// TIA Portal project "Flaconneuse" (V16)

(* hardware
DEVICE "Station S71500/ET200MP_1"  S7-1500 station
   slot 0: "Châssis_0"  Rack  6ES7 590-1***0-0AA0
   slot 0: "PM 70W 120/230VAC"  PM 70W 120/230VAC  6EP1332-4BA00
   slot 1: "PLC_1"  CPU 1511-1 PN  6ES7 511-1AK02-0AB0  V2.8
      slot 3: "Ecran CPU_1"  6ES7591-1AA00-0AA0
      slot 32768: "Interface PROFINET_1"  X1
         slot 32769: "Port_1"  X1 P1
         slot 32770: "Port_2"  X1 P2
      slot 34817: "Virtual CP interface port_1"  Virtual CP interface port  Virtual CP interface port
   slot 2: "DI 32x24VDC BA_1"  DI 32x24VDC BA  6ES7 521-1BL10-0AA0  V1.0
   slot 3: "DQ 32x24VDC/0.5A BA_1"  DQ 32x24VDC/0.5A BA  6ES7 522-1BL10-0AA0  V1.0
   slot 4: "CM 1542-5_1"  CM 1542-5  6GK7 542-5DX00-0XE0  V1.0
*)

// ===== PLC "PLC_1"  CPU 1511-1 PN =====

VAR_GLOBAL   // PLC tag table "Table de variables standard"
   "Marche cycle" AT %I0.0 : Bool;
   "Arret cycle" AT %I0.1 : Bool;
   "Selecteur sur Auto" AT %I0.3 : Bool;
   "Selecteur sur Manu" AT %I0.4 : Bool;
   "BP Manu" AT %I0.5 : Bool;
   "BP Purge" AT %I0.6 : Bool;
   "S1 pa" AT %I1.0 : Bool;   // Flacon en entree
   "S2 t0" AT %I1.1 : Bool;   // Verin de transfert rentre
   "S3 t1" AT %I1.2 : Bool;   // Verin de transfert sorti
   "S4 e1" AT %I1.3 : Bool;   // Verin d entrainement sorti
   "S5 i1" AT %I1.4 : Bool;   // Verin d indexage sorti
   "S6 p1" AT %I1.5 : Bool;   // Pompe sorti
   "S7 p0" AT %I1.6 : Bool;   // Pompe rentree
   "S8 r0" AT %I1.7 : Bool;   // Verin de vissage en bas
   "S9 r1" AT %I2.0 : Bool;   // Verin de vissage en haut
   "S10 b" AT %I2.1 : Bool;   // Flacon maintenu
   "S11 bour" AT %I2.2 : Bool;   // Bourage en sortie
   "S12 pr" AT %I2.3 : Bool;   // Presence remplissage
   "Voyant defaut" AT %Q0.0 : Bool;
   "EV1 T-" AT %Q0.1 : Bool;   // Rentrer verin transfert
   "EV2 T+" AT %Q0.2 : Bool;   // Sortir verin transfert
   "EV3 E-" AT %Q0.3 : Bool;   // Rentrer verin entrainement
   "EV4 I-" AT %Q0.4 : Bool;   // Rentrer verin indexage
   "EV5 P+" AT %Q0.5 : Bool;   // Sortir pompe
   "EV6 P-" AT %Q0.6 : Bool;   // Rentrer pompe
   "EV7 A" AT %Q0.7 : Bool;   // Commande arrivee liquide
   "EV8 J" AT %Q1.0 : Bool;   // Commande sortie liquide
   "EV9 B+" AT %Q1.1 : Bool;   // Maintenir flacon
   "EV10 R+" AT %Q1.2 : Bool;   // Descendre vissage
   "KM1" AT %Q1.4 : Bool;   // Moteur tapis
   "KM2" AT %Q1.5 : Bool;   // Moteur visseuse
   "IndexPlateau" AT %MW200 : Int;   // Les trois premiers bits de ce mot servent à savoir si il y a (ou non) un flacon sous chacun des postes
   "FM_FinPlateau" AT %M100.0 : Bool;
   "CI" AT %M120.0 : Bool;   // Condition initiales ok
   "DefautActif" AT %MW300 : Word;
END_VAR

DATA_BLOCK "X30_TournerPlateau_DB"   // DB1
{ S7_Optimized_Access := 'TRUE' }
VERSION : 0.1
// stored: InstanceOfName X30_TournerPlateau
"X30_TournerPlateau"
BEGIN
END_DATA_BLOCK

DATA_BLOCK "Sorties_DB"   // DB2
{ S7_Optimized_Access := 'TRUE' }
VERSION : 0.1
// stored: InstanceOfName Sorties
"Sorties"
BEGIN
END_DATA_BLOCK

DATA_BLOCK "X100_Remplir_DB"   // DB3
{ S7_Optimized_Access := 'TRUE' }
VERSION : 0.1
// stored: InstanceOfName X100_Remplir
"X100_Remplir"
BEGIN
END_DATA_BLOCK

DATA_BLOCK "X130_Visser_DB"   // DB4
{ S7_Optimized_Access := 'TRUE' }
VERSION : 0.1
// stored: InstanceOfName X130_Visser
"X130_Visser"
BEGIN
END_DATA_BLOCK

DATA_BLOCK "X160_Evacuer_DB"   // DB5
{ S7_Optimized_Access := 'TRUE' }
VERSION : 0.1
// stored: InstanceOfName X160_Evacuer
"X160_Evacuer"
BEGIN
END_DATA_BLOCK

DATA_BLOCK "X10_Conduite_DB"   // DB6
{ S7_Optimized_Access := 'TRUE' }
VERSION : 0.1
// stored: InstanceOfName X10_Conduite
"X10_Conduite"
BEGIN
END_DATA_BLOCK

DATA_BLOCK "X500_ModesDeMarche_DB"   // DB7
{ S7_Optimized_Access := 'TRUE' }
VERSION : 0.1
// stored: InstanceOfName X500_ModesDeMarche
"X500_ModesDeMarche"
BEGIN
END_DATA_BLOCK

DATA_BLOCK "GestionIndexPlateau_DB"   // DB8
{ S7_Optimized_Access := 'TRUE' }
VERSION : 0.1
// stored: InstanceOfName GestionIndexPlateau
"GestionIndexPlateau"
BEGIN
END_DATA_BLOCK

DATA_BLOCK "CondInitiales_DB"   // DB9
{ S7_Optimized_Access := 'TRUE' }
VERSION : 0.1
// stored: InstanceOfName CondInitiales
"CondInitiales"
BEGIN
END_DATA_BLOCK

DATA_BLOCK "defauts_DB"   // DB12
{ S7_Optimized_Access := 'TRUE' }
VERSION : 0.1
// stored: InstanceOfName defauts
"defauts"
BEGIN
END_DATA_BLOCK

// folder: System blocks/Program resources

DATA_BLOCK "IEC_Timer_0_DB"   // DB10
{ S7_Optimized_Access := 'TRUE' }
AUTHOR : Simatic
FAMILY : IEC
NAME : IEC_TMR
VERSION : 1.0
// stored: InstanceOfName IEC_TIMER
"IEC_TIMER"
BEGIN
END_DATA_BLOCK

DATA_BLOCK "IEC_Timer_0_DB_1"   // DB11
{ S7_Optimized_Access := 'TRUE' }
AUTHOR : Simatic
FAMILY : IEC
NAME : IEC_TMR
VERSION : 1.0
// stored: InstanceOfName IEC_TIMER
"IEC_TIMER"
BEGIN
END_DATA_BLOCK

// folder: (top level)

FUNCTION_BLOCK "X30_TournerPlateau"   // FB1, GRAPH_PLUS
{ S7_Optimized_Access := 'TRUE' }
VERSION : 0.1
   VAR_INPUT
      OFF_SQ : Bool := false;   // Désactiver le graphe
      INIT_SQ : Bool := false;   // Mettre le graphe à l'état initial
      ACK_EF : Bool := false;   // Acquitter toutes les erreurs et perturbations
      S_PREV : Bool := false;   // Afficher l'étape précédente dans le paramètre S_NO
      S_NEXT : Bool := false;   // Afficher l'étape suivante dans le paramètre S_NO
      SW_AUTO : Bool := false;   // Mode automatique
      SW_TAP : Bool := false;   // Mode semi-automatique/Activation de l'étape suivante avec transition
      SW_TOP : Bool := false;   // Mode semi-automatique/Ignorer la transition
      SW_MAN : Bool := false;   // Mode manuel
      S_SEL : Int := 0;   // Sélectionner l'étape à afficher dans S_NO
      S_ON : Bool := false;   // Activer l'étape figurant dans le paramètre S_NO
      S_OFF : Bool := false;   // Désactiver l'étape figurant dans le paramètre S_NO
      T_PUSH : Bool := false;   // Validation de commutation pour transition en mode semi-automatique
   END_VAR
   VAR_OUTPUT
      S_NO : Int := 0;   // Numéro d'étape
      S_MORE : Bool := false;   // Il existe d'autres étapes qui peuvent être affichées dans S_NO.
      S_ACTIVE : Bool := false;   // L'étape affichée dans le paramètre S_NO est activée
      ERR_FLT : Bool := false;   // Erreur groupée Interlock or Supervision
      AUTO_ON : Bool := false;   // Mode automatique activé
      TAP_ON : Bool := false;   // Mode semi-automatique/Etape avec transition activé
      TOP_ON : Bool := false;   // Mode semi-automatique/Ignorer la transition activé
      MAN_ON : Bool := false;   // Mode manuel activé
   END_VAR
   VAR
      HMI_INFO : Array[0..8] of UInt;
      IF_PAR : G7_IfParPlus_V6;
      RT_DATA : G7_RTDataPlus_V6;   // Plage de données interne
      Trans1 : G7_TransitionPlus_V6;   // Structure de la transition
      Trans2 : G7_TransitionPlus_V6;   // Structure de la transition
      Trans3 : G7_TransitionPlus_V6;   // Structure de la transition
      Trans4 : G7_TransitionPlus_V6;   // Structure de la transition
      Trans5 : G7_TransitionPlus_V6;   // Structure de la transition
      Trans6 : G7_TransitionPlus_V6;   // Structure de la transition
      Trans7 : G7_TransitionPlus_V6;   // Structure de la transition
      Trans8 : G7_TransitionPlus_V6;   // Structure de la transition
      Step30 : G7_StepPlus_V6;   // Structure de l'étape
      Step32 : G7_StepPlus_V6;   // Structure de l'étape
      Step34 : G7_StepPlus_V6;   // Structure de l'étape
      Step36 : G7_StepPlus_V6;   // Structure de l'étape
      Step38 : G7_StepPlus_V6;   // Structure de l'étape
      Step40 : G7_StepPlus_V6;   // Structure de l'étape
      Step42 : G7_StepPlus_V6;   // Structure de l'étape
      Step44 : G7_StepPlus_V6;   // Structure de l'étape
      SINI : Array[0..1] of USInt;
      LSTT : Array[0..7] of USInt;
      ATAJ : Array[0..7] of USInt;
      ATAB : Array[0..7] of USInt;
      PSTT : Array[0..7] of USInt;
      NSTT : Array[0..7] of USInt;
      ASSJ : Array[0..7] of USInt;
      ASSB : Array[0..7] of USInt;
      PTTS : Array[0..7] of USInt;
      NTTS : Array[0..7] of USInt;
      SW_SQTS : Array[0..7] of USInt;
      SWITCH : Array[0..0] of USInt;
      TVX : Array[0..1] of USInt;
      TTX : Array[0..1] of USInt;
      TSX : Array[0..1] of USInt;
      S00X : Array[0..1] of USInt;
      SOFFX : Array[0..1] of USInt;
      SONX : Array[0..1] of USInt;
      SAX : Array[0..1] of USInt;
      SERRX : Array[0..8] of USInt;
      SMX : Array[0..8] of USInt;
      S0X : Array[0..8] of USInt;
      S1X : Array[0..8] of USInt;
      IL_ALARM_INST : Diag_Alarm;
      SUP_ALARM_INST : Diag_Alarm;
      STEP_TIME_ALARM_INST : Diag_Alarm;
      IEC_TIMER_INST : IEC_TIMER;
      TRANSACTION_FLAG : Bool := false;
   END_VAR
   // SINI[0] := 2;
   // LSTT[0] := 255;
   // LSTT[1] := 255;
   // LSTT[2] := 255;
   // LSTT[3] := 255;
   // LSTT[4] := 255;
   // LSTT[5] := 255;
   // LSTT[6] := 255;
   // ATAJ[1] := 1;
   // ATAJ[2] := 2;
   // ATAJ[3] := 3;
   // ATAJ[4] := 4;
   // ATAJ[5] := 5;
   // ATAJ[6] := 6;
   // ATAJ[7] := 7;
   // ATAB[1] := 1;
   // ATAB[2] := 2;
   // ATAB[3] := 3;
   // ATAB[4] := 4;
   // ATAB[5] := 5;
   // ATAB[6] := 6;
   // ATAB[7] := 7;
   // PSTT[1] := 1;
   // PSTT[2] := 2;
   // PSTT[3] := 3;
   // PSTT[4] := 4;
   // PSTT[5] := 5;
   // PSTT[6] := 6;
   // PSTT[7] := 7;
   // NSTT[0] := 1;
   // NSTT[1] := 2;
   // NSTT[2] := 3;
   // NSTT[3] := 4;
   // NSTT[4] := 5;
   // NSTT[5] := 6;
   // NSTT[6] := 7;
   // ASSJ[1] := 1;
   // ASSJ[2] := 2;
   // ASSJ[3] := 3;
   // ASSJ[4] := 4;
   // ASSJ[5] := 5;
   // ASSJ[6] := 6;
   // ASSJ[7] := 7;
   // ASSB[1] := 1;
   // ASSB[2] := 2;
   // ASSB[3] := 3;
   // ASSB[4] := 4;
   // ASSB[5] := 5;
   // ASSB[6] := 6;
   // ASSB[7] := 7;
   // PTTS[0] := 255;
   // PTTS[2] := 1;
   // PTTS[3] := 2;
   // PTTS[4] := 3;
   // PTTS[5] := 4;
   // PTTS[6] := 5;
   // PTTS[7] := 6;
   // NTTS[1] := 1;
   // NTTS[2] := 2;
   // NTTS[3] := 3;
   // NTTS[4] := 4;
   // NTTS[5] := 5;
   // NTTS[6] := 6;
   // NTTS[7] := 7;
   // TVX[0] := 16#1;
   // TTX[0] := 16#1;
   // TSX[0] := 16#1;
   // S00X[0] := 16#1;
   // SOFFX[0] := 16#1;
   // SONX[0] := 16#1;
   // SAX[0] := 16#1;
   // SERRX[0] := 16#1;
   // SMX[0] := 16#1;
   // S0X[0] := 16#1;
   // S1X[0] := 16#1;
BEGIN
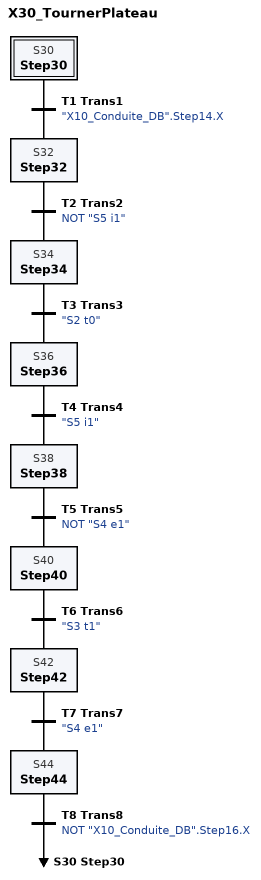
   // sequencer 1
   INITIAL_STEP Step30:   // S30, max time T#10S, warning time T#7S
   END_STEP
   TRANSITION Trans1 FROM Step30 TO Step32   // T1
      := "X10_Conduite_DB".Step14.X;
   END_TRANSITION
   STEP Step32:   // S32, max time T#10S, warning time T#7S
   END_STEP
   TRANSITION Trans2 FROM Step32 TO Step34   // T2: Vérin indexage rentré
      := NOT "S5 i1";
   END_TRANSITION
   STEP Step34:   // S34, max time T#10S, warning time T#7S
   END_STEP
   TRANSITION Trans3 FROM Step34 TO Step36   // T3: Vérin transfert rentré
      := "S2 t0";
   END_TRANSITION
   STEP Step36:   // S36, max time T#10S, warning time T#7S
   END_STEP
   TRANSITION Trans4 FROM Step36 TO Step38   // T4: vérin indexage sorti
      := "S5 i1";
   END_TRANSITION
   STEP Step38:   // S38, max time T#10S, warning time T#7S
   END_STEP
   TRANSITION Trans5 FROM Step38 TO Step40   // T5: Vérin entrainement rentré
      := NOT "S4 e1";
   END_TRANSITION
   STEP Step40:   // S40, max time T#10S, warning time T#7S
   END_STEP
   TRANSITION Trans6 FROM Step40 TO Step42   // T6: Vérin transfert sorti
      := "S3 t1";
   END_TRANSITION
   STEP Step42:   // S42, max time T#10S, warning time T#7S
   END_STEP
   TRANSITION Trans7 FROM Step42 TO Step44   // T7: Vérin entrainement sorti
      := "S4 e1";
   END_TRANSITION
   STEP Step44:   // S44, max time T#10S, warning time T#7S
   END_STEP
   TRANSITION Trans8 FROM Step44 TO Step30   // T8, jump
      := NOT "X10_Conduite_DB".Step16.X;
   END_TRANSITION
END_FUNCTION_BLOCK

FUNCTION_BLOCK "Sorties"   // FB2, LAD
{ S7_Optimized_Access := 'TRUE' }
VERSION : 0.1
BEGIN

REGION Network 1: Rentrer verin transfert
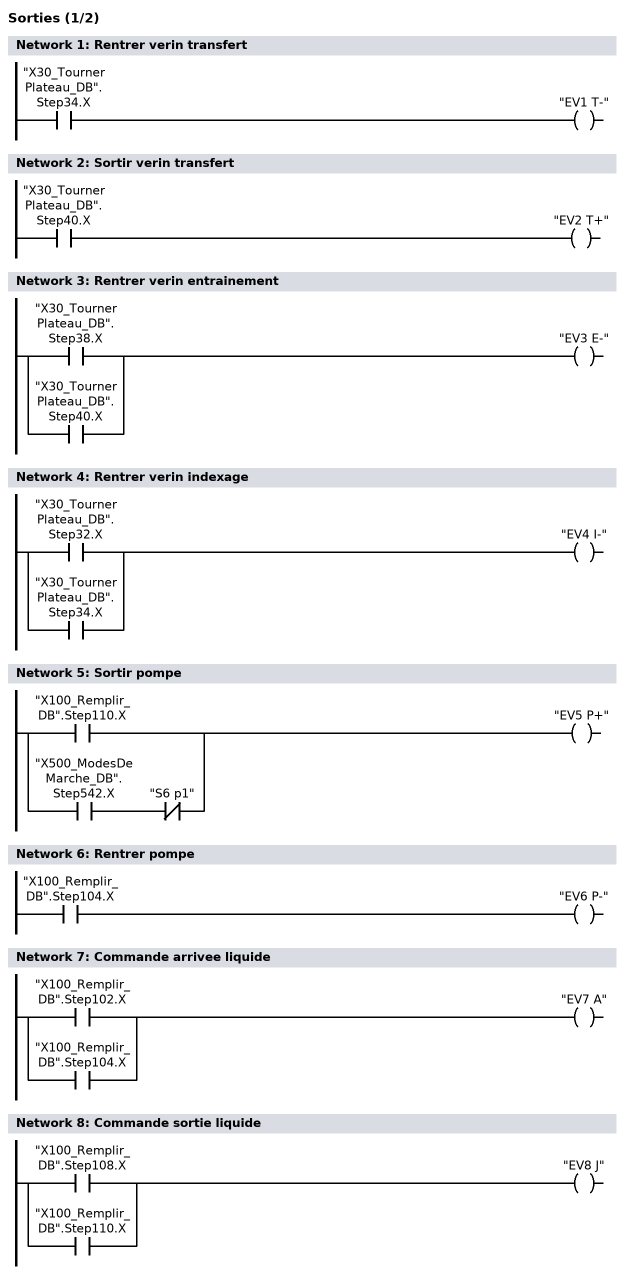
   RUNG wire#powerrail
      Contact( "X30_TournerPlateau_DB".Step34.X )
      Coil( "EV1 T-" )
   END_RUNG
   // the same network as SCL:
   "EV1 T-" := "X30_TournerPlateau_DB".Step34.X;
END_REGION

REGION Network 2: Sortir verin transfert
   RUNG wire#powerrail
      Contact( "X30_TournerPlateau_DB".Step40.X )
      Coil( "EV2 T+" )
   END_RUNG
   // the same network as SCL:
   "EV2 T+" := "X30_TournerPlateau_DB".Step40.X;
END_REGION

REGION Network 3: Rentrer verin entrainement
   RUNG wire#powerrail
      Contact( "X30_TournerPlateau_DB".Step38.X )
      wire#w1
      Coil( "EV3 E-" )
   END_RUNG
   RUNG wire#powerrail
      Contact( "X30_TournerPlateau_DB".Step40.X )
   END_RUNG wire#w1
   // the same network as SCL:
   "EV3 E-" := "X30_TournerPlateau_DB".Step38.X OR "X30_TournerPlateau_DB".Step40.X;
END_REGION

REGION Network 4: Rentrer verin indexage
   RUNG wire#powerrail
      Contact( "X30_TournerPlateau_DB".Step32.X )
      wire#w1
      Coil( "EV4 I-" )
   END_RUNG
   RUNG wire#powerrail
      Contact( "X30_TournerPlateau_DB".Step34.X )
   END_RUNG wire#w1
   // the same network as SCL:
   "EV4 I-" := "X30_TournerPlateau_DB".Step32.X OR "X30_TournerPlateau_DB".Step34.X;
END_REGION

REGION Network 5: Sortir pompe
   RUNG wire#powerrail
      Contact( "X100_Remplir_DB".Step110.X )
      wire#w1
      Coil( "EV5 P+" )
   END_RUNG
   RUNG wire#powerrail
      Contact( "X500_ModesDeMarche_DB".Step542.X )
      I_Contact( "S6 p1" )
   END_RUNG wire#w1
   // the same network as SCL:
   "EV5 P+" := "X100_Remplir_DB".Step110.X OR ("X500_ModesDeMarche_DB".Step542.X AND NOT "S6 p1");
END_REGION

REGION Network 6: Rentrer pompe
   RUNG wire#powerrail
      Contact( "X100_Remplir_DB".Step104.X )
      Coil( "EV6 P-" )
   END_RUNG
   // the same network as SCL:
   "EV6 P-" := "X100_Remplir_DB".Step104.X;
END_REGION

REGION Network 7: Commande arrivee liquide
   RUNG wire#powerrail
      Contact( "X100_Remplir_DB".Step102.X )
      wire#w1
      Coil( "EV7 A" )
   END_RUNG
   RUNG wire#powerrail
      Contact( "X100_Remplir_DB".Step104.X )
   END_RUNG wire#w1
   // the same network as SCL:
   "EV7 A" := "X100_Remplir_DB".Step102.X OR "X100_Remplir_DB".Step104.X;
END_REGION

REGION Network 8: Commande sortie liquide
   RUNG wire#powerrail
      Contact( "X100_Remplir_DB".Step108.X )
      wire#w1
      Coil( "EV8 J" )
   END_RUNG
   RUNG wire#powerrail
      Contact( "X100_Remplir_DB".Step110.X )
   END_RUNG wire#w1
   // the same network as SCL:
   "EV8 J" := "X100_Remplir_DB".Step108.X OR "X100_Remplir_DB".Step110.X;
END_REGION

REGION Network 9: Maintenir flacon
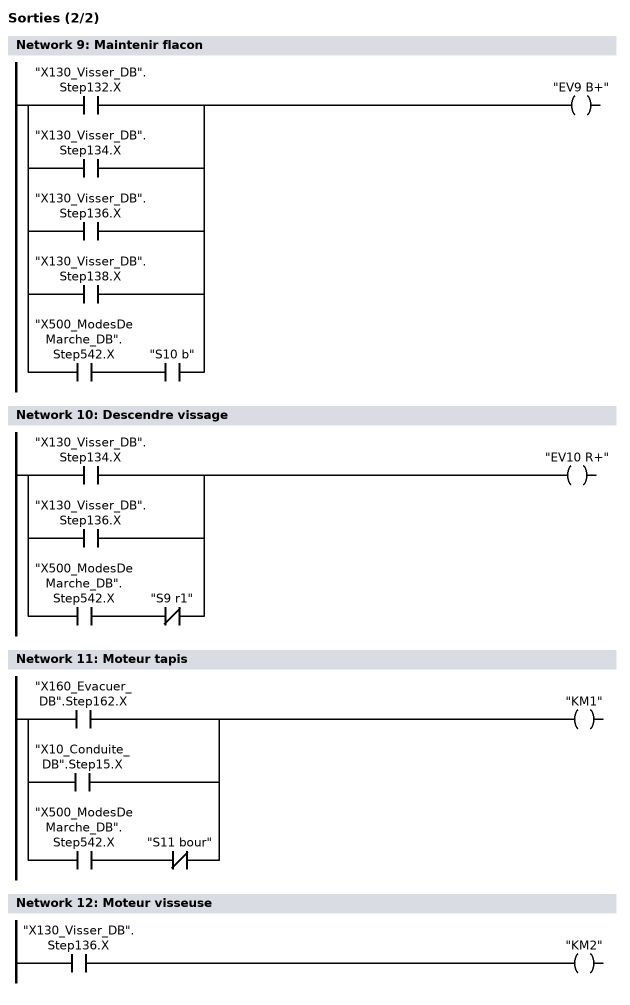
   RUNG wire#powerrail
      Contact( "X130_Visser_DB".Step132.X )
      wire#w1
      Coil( "EV9 B+" )
   END_RUNG
   RUNG wire#powerrail
      Contact( "X130_Visser_DB".Step134.X )
   END_RUNG wire#w1
   RUNG wire#powerrail
      Contact( "X130_Visser_DB".Step136.X )
   END_RUNG wire#w1
   RUNG wire#powerrail
      Contact( "X130_Visser_DB".Step138.X )
   END_RUNG wire#w1
   RUNG wire#powerrail
      Contact( "X500_ModesDeMarche_DB".Step542.X )
      Contact( "S10 b" )
   END_RUNG wire#w1
   // the same network as SCL:
   "EV9 B+" := "X130_Visser_DB".Step132.X OR "X130_Visser_DB".Step134.X OR "X130_Visser_DB".Step136.X OR "X130_Visser_DB".Step138.X OR ("X500_ModesDeMarche_DB".Step542.X AND "S10 b");
END_REGION

REGION Network 10: Descendre vissage
   RUNG wire#powerrail
      Contact( "X130_Visser_DB".Step134.X )
      wire#w1
      Coil( "EV10 R+" )
   END_RUNG
   RUNG wire#powerrail
      Contact( "X130_Visser_DB".Step136.X )
   END_RUNG wire#w1
   RUNG wire#powerrail
      Contact( "X500_ModesDeMarche_DB".Step542.X )
      I_Contact( "S9 r1" )
   END_RUNG wire#w1
   // the same network as SCL:
   "EV10 R+" := "X130_Visser_DB".Step134.X OR "X130_Visser_DB".Step136.X OR ("X500_ModesDeMarche_DB".Step542.X AND NOT "S9 r1");
END_REGION

REGION Network 11: Moteur tapis
   RUNG wire#powerrail
      Contact( "X160_Evacuer_DB".Step162.X )
      wire#w1
      Coil( "KM1" )
   END_RUNG
   RUNG wire#powerrail
      Contact( "X10_Conduite_DB".Step15.X )
   END_RUNG wire#w1
   RUNG wire#powerrail
      Contact( "X500_ModesDeMarche_DB".Step542.X )
      I_Contact( "S11 bour" )
   END_RUNG wire#w1
   // the same network as SCL:
   "KM1" := "X160_Evacuer_DB".Step162.X OR "X10_Conduite_DB".Step15.X OR ("X500_ModesDeMarche_DB".Step542.X AND NOT "S11 bour");
END_REGION

REGION Network 12: Moteur visseuse
   RUNG wire#powerrail
      Contact( "X130_Visser_DB".Step136.X )
      Coil( "KM2" )
   END_RUNG
   // the same network as SCL:
   "KM2" := "X130_Visser_DB".Step136.X;
END_REGION
END_FUNCTION_BLOCK

FUNCTION_BLOCK "X100_Remplir"   // FB3, GRAPH_PLUS
{ S7_Optimized_Access := 'TRUE' }
VERSION : 0.1
   VAR_INPUT
      OFF_SQ : Bool := false;   // Désactiver le graphe
      INIT_SQ : Bool := false;   // Mettre le graphe à l'état initial
      ACK_EF : Bool := false;   // Acquitter toutes les erreurs et perturbations
      S_PREV : Bool := false;   // Afficher l'étape précédente dans le paramètre S_NO
      S_NEXT : Bool := false;   // Afficher l'étape suivante dans le paramètre S_NO
      SW_AUTO : Bool := false;   // Mode automatique
      SW_TAP : Bool := false;   // Mode semi-automatique/Activation de l'étape suivante avec transition
      SW_TOP : Bool := false;   // Mode semi-automatique/Ignorer la transition
      SW_MAN : Bool := false;   // Mode manuel
      S_SEL : Int := 0;   // Sélectionner l'étape à afficher dans S_NO
      S_ON : Bool := false;   // Activer l'étape figurant dans le paramètre S_NO
      S_OFF : Bool := false;   // Désactiver l'étape figurant dans le paramètre S_NO
      T_PUSH : Bool := false;   // Validation de commutation pour transition en mode semi-automatique
   END_VAR
   VAR_OUTPUT
      S_NO : Int := 0;   // Numéro d'étape
      S_MORE : Bool := false;   // Il existe d'autres étapes qui peuvent être affichées dans S_NO.
      S_ACTIVE : Bool := false;   // L'étape affichée dans le paramètre S_NO est activée
      ERR_FLT : Bool := false;   // Erreur groupée Interlock or Supervision
      AUTO_ON : Bool := false;   // Mode automatique activé
      TAP_ON : Bool := false;   // Mode semi-automatique/Etape avec transition activé
      TOP_ON : Bool := false;   // Mode semi-automatique/Ignorer la transition activé
      MAN_ON : Bool := false;   // Mode manuel activé
   END_VAR
   VAR
      HMI_INFO : Array[0..8] of UInt;
      IF_PAR : G7_IfParPlus_V6;
      RT_DATA : G7_RTDataPlus_V6;   // Plage de données interne
      Trans2 : G7_TransitionPlus_V6;   // Structure de la transition
      Trans3 : G7_TransitionPlus_V6;   // Structure de la transition
      Trans4 : G7_TransitionPlus_V6;   // Structure de la transition
      Trans5 : G7_TransitionPlus_V6;   // Structure de la transition
      Trans6 : G7_TransitionPlus_V6;   // Structure de la transition
      Trans7 : G7_TransitionPlus_V6;   // Structure de la transition
      Trans8 : G7_TransitionPlus_V6;   // Structure de la transition
      Trans9 : G7_TransitionPlus_V6;   // Structure de la transition
      Step100 : G7_StepPlus_V6;   // Structure de l'étape
      Step102 : G7_StepPlus_V6;   // Structure de l'étape
      Step104 : G7_StepPlus_V6;   // Structure de l'étape
      Step106 : G7_StepPlus_V6;   // Structure de l'étape
      Step108 : G7_StepPlus_V6;   // Structure de l'étape
      Step110 : G7_StepPlus_V6;   // Structure de l'étape
      Step112 : G7_StepPlus_V6;   // Structure de l'étape
      SINI : Array[0..1] of USInt;
      LSTT : Array[0..7] of USInt;
      ATAJ : Array[0..7] of USInt;
      ATAB : Array[0..7] of USInt;
      PSTT : Array[0..7] of USInt;
      NSTT : Array[0..7] of USInt;
      ASSJ : Array[0..6] of USInt;
      ASSB : Array[0..6] of USInt;
      PTTS : Array[0..6] of USInt;
      NTTS : Array[0..6] of USInt;
      SW_SQTS : Array[0..6] of USInt;
      SWITCH : Array[0..1] of USInt;
      TVX : Array[0..3] of USInt;
      TTX : Array[0..3] of USInt;
      TSX : Array[0..1] of USInt;
      S00X : Array[0..1] of USInt;
      SOFFX : Array[0..1] of USInt;
      SONX : Array[0..1] of USInt;
      SAX : Array[0..1] of USInt;
      SERRX : Array[0..7] of USInt;
      SMX : Array[0..7] of USInt;
      S0X : Array[0..7] of USInt;
      S1X : Array[0..7] of USInt;
      IL_ALARM_INST : Diag_Alarm;
      SUP_ALARM_INST : Diag_Alarm;
      STEP_TIME_ALARM_INST : Diag_Alarm;
      IEC_TIMER_INST : IEC_TIMER;
      TRANSACTION_FLAG : Bool := false;
   END_VAR
   // SINI[0] := 2;
   // LSTT[0] := 255;
   // LSTT[1] := 255;
   // LSTT[2] := 255;
   // LSTT[3] := 255;
   // LSTT[4] := 255;
   // LSTT[6] := 255;
   // ATAJ[1] := 1;
   // ATAJ[2] := 2;
   // ATAJ[3] := 3;
   // ATAJ[4] := 6;
   // ATAJ[5] := 5;
   // ATAJ[6] := 4;
   // ATAB[1] := 1;
   // ATAB[2] := 2;
   // ATAB[3] := 3;
   // ATAB[4] := 4;
   // ATAB[5] := 5;
   // ATAB[6] := 7;
   // PSTT[1] := 2;
   // PSTT[2] := 3;
   // PSTT[3] := 4;
   // PSTT[4] := 5;
   // PSTT[5] := 6;
   // NSTT[7] := 1;
   // NSTT[0] := 2;
   // NSTT[1] := 3;
   // NSTT[2] := 4;
   // NSTT[3] := 5;
   // NSTT[4] := 6;
   // NSTT[6] := 6;
   // ASSJ[1] := 1;
   // ASSJ[2] := 2;
   // ASSJ[3] := 3;
   // ASSJ[4] := 4;
   // ASSJ[5] := 5;
   // ASSJ[6] := 6;
   // ASSB[1] := 1;
   // ASSB[2] := 2;
   // ASSB[3] := 3;
   // ASSB[4] := 4;
   // ASSB[5] := 5;
   // ASSB[6] := 6;
   // PTTS[0] := 255;
   // NTTS[0] := 7;
   // PTTS[3] := 1;
   // PTTS[4] := 2;
   // PTTS[5] := 3;
   // PTTS[6] := 4;
   // SW_SQTS[1] := 1;
   // NTTS[2] := 1;
   // NTTS[3] := 2;
   // NTTS[4] := 3;
   // NTTS[5] := 4;
   // NTTS[6] := 5;
   // TVX[0] := 16#1;
   // TTX[0] := 16#1;
   // TSX[0] := 16#1;
   // S00X[0] := 16#1;
   // SOFFX[0] := 16#1;
   // SONX[0] := 16#1;
   // SAX[0] := 16#1;
   // SERRX[0] := 16#1;
   // SMX[0] := 16#1;
   // S0X[0] := 16#1;
   // S1X[0] := 16#1;
   // LSTT[7] := 255;
   // ATAJ[7] := 7;
   // ATAB[7] := 6;
   // PSTT[0] := 1;
   // PTTS[1] := 7;
   // SW_SQTS[2] := 1;
   // SW_SQTS[3] := 1;
   // SW_SQTS[4] := 1;
   // SW_SQTS[5] := 1;
   // SW_SQTS[6] := 2;
BEGIN
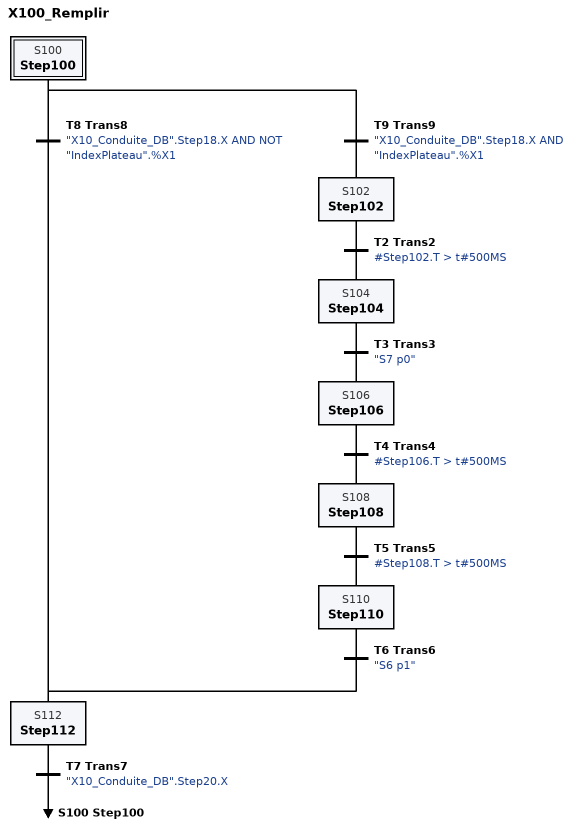
   // sequencer 1
   INITIAL_STEP Step100:   // S100, max time T#10S, warning time T#7S
   END_STEP
   TRANSITION Trans8 FROM Step100 TO Step112   // T8
      := "X10_Conduite_DB".Step18.X AND NOT "IndexPlateau".%X1;
   END_TRANSITION
   TRANSITION Trans9 FROM Step100 TO Step102   // T9
      := "X10_Conduite_DB".Step18.X AND "IndexPlateau".%X1;
   END_TRANSITION
   STEP Step102:   // S102, max time T#10S, warning time T#7S
   END_STEP
   TRANSITION Trans2 FROM Step102 TO Step104   // T2: Arrivée de liquide ouverte
      := #Step102.T > t#500MS;
   END_TRANSITION
   STEP Step104:   // S104, max time T#10S, warning time T#7S
   END_STEP
   TRANSITION Trans3 FROM Step104 TO Step106   // T3: Pompe rentrée
      := "S7 p0";
   END_TRANSITION
   STEP Step106:   // S106, max time T#10S, warning time T#7S
   END_STEP
   TRANSITION Trans4 FROM Step106 TO Step108   // T4: Arrivée de liquide fermée
      := #Step106.T > t#500MS;
   END_TRANSITION
   STEP Step108:   // S108, max time T#10S, warning time T#7S
   END_STEP
   TRANSITION Trans5 FROM Step108 TO Step110   // T5: Sortie de liquide ouverte
      := #Step108.T > t#500MS;
   END_TRANSITION
   STEP Step110:   // S110, max time T#10S, warning time T#7S
   END_STEP
   TRANSITION Trans6 FROM Step110 TO Step112   // T6: Pompe sortie
      := "S6 p1";
   END_TRANSITION
   STEP Step112:   // S112, max time T#10S, warning time T#7S
   END_STEP
   TRANSITION Trans7 FROM Step112 TO Step100   // T7, jump
      := "X10_Conduite_DB".Step20.X;
   END_TRANSITION
END_FUNCTION_BLOCK

FUNCTION_BLOCK "X130_Visser"   // FB4, GRAPH_PLUS
{ S7_Optimized_Access := 'TRUE' }
VERSION : 0.1
   VAR_INPUT
      OFF_SQ : Bool := false;   // Désactiver le graphe
      INIT_SQ : Bool := false;   // Mettre le graphe à l'état initial
      ACK_EF : Bool := false;   // Acquitter toutes les erreurs et perturbations
      S_PREV : Bool := false;   // Afficher l'étape précédente dans le paramètre S_NO
      S_NEXT : Bool := false;   // Afficher l'étape suivante dans le paramètre S_NO
      SW_AUTO : Bool := false;   // Mode automatique
      SW_TAP : Bool := false;   // Mode semi-automatique/Activation de l'étape suivante avec transition
      SW_TOP : Bool := false;   // Mode semi-automatique/Ignorer la transition
      SW_MAN : Bool := false;   // Mode manuel
      S_SEL : Int := 0;   // Sélectionner l'étape à afficher dans S_NO
      S_ON : Bool := false;   // Activer l'étape figurant dans le paramètre S_NO
      S_OFF : Bool := false;   // Désactiver l'étape figurant dans le paramètre S_NO
      T_PUSH : Bool := false;   // Validation de commutation pour transition en mode semi-automatique
   END_VAR
   VAR_OUTPUT
      S_NO : Int := 0;   // Numéro d'étape
      S_MORE : Bool := false;   // Il existe d'autres étapes qui peuvent être affichées dans S_NO.
      S_ACTIVE : Bool := false;   // L'étape affichée dans le paramètre S_NO est activée
      ERR_FLT : Bool := false;   // Erreur groupée Interlock or Supervision
      AUTO_ON : Bool := false;   // Mode automatique activé
      TAP_ON : Bool := false;   // Mode semi-automatique/Etape avec transition activé
      TOP_ON : Bool := false;   // Mode semi-automatique/Ignorer la transition activé
      MAN_ON : Bool := false;   // Mode manuel activé
   END_VAR
   VAR
      HMI_INFO : Array[0..8] of UInt;
      IF_PAR : G7_IfParPlus_V6;
      RT_DATA : G7_RTDataPlus_V6;   // Plage de données interne
      Trans1 : G7_TransitionPlus_V6;   // Structure de la transition
      Trans2 : G7_TransitionPlus_V6;   // Structure de la transition
      Trans3 : G7_TransitionPlus_V6;   // Structure de la transition
      Trans4 : G7_TransitionPlus_V6;   // Structure de la transition
      Trans5 : G7_TransitionPlus_V6;   // Structure de la transition
      Trans6 : G7_TransitionPlus_V6;   // Structure de la transition
      Trans7 : G7_TransitionPlus_V6;   // Structure de la transition
      Step130 : G7_StepPlus_V6;   // Structure de l'étape
      Step132 : G7_StepPlus_V6;   // Structure de l'étape
      Step134 : G7_StepPlus_V6;   // Structure de l'étape
      Step136 : G7_StepPlus_V6;   // Structure de l'étape
      Step138 : G7_StepPlus_V6;   // Structure de l'étape
      Step140 : G7_StepPlus_V6;   // Structure de l'étape
      SINI : Array[0..1] of USInt;
      LSTT : Array[0..6] of USInt;
      ATAJ : Array[0..6] of USInt;
      ATAB : Array[0..6] of USInt;
      PSTT : Array[0..6] of USInt;
      NSTT : Array[0..6] of USInt;
      ASSJ : Array[0..5] of USInt;
      ASSB : Array[0..5] of USInt;
      PTTS : Array[0..5] of USInt;
      NTTS : Array[0..5] of USInt;
      SW_SQTS : Array[0..5] of USInt;
      SWITCH : Array[0..1] of USInt;
      TVX : Array[0..3] of USInt;
      TTX : Array[0..3] of USInt;
      TSX : Array[0..1] of USInt;
      S00X : Array[0..1] of USInt;
      SOFFX : Array[0..1] of USInt;
      SONX : Array[0..1] of USInt;
      SAX : Array[0..1] of USInt;
      SERRX : Array[0..6] of USInt;
      SMX : Array[0..6] of USInt;
      S0X : Array[0..6] of USInt;
      S1X : Array[0..6] of USInt;
      IL_ALARM_INST : Diag_Alarm;
      SUP_ALARM_INST : Diag_Alarm;
      STEP_TIME_ALARM_INST : Diag_Alarm;
      IEC_TIMER_INST : IEC_TIMER;
      TRANSACTION_FLAG : Bool := false;
   END_VAR
   // SINI[0] := 2;
   // LSTT[0] := 255;
   // LSTT[1] := 255;
   // LSTT[2] := 255;
   // LSTT[3] := 255;
   // LSTT[4] := 255;
   // ATAJ[1] := 1;
   // ATAJ[2] := 2;
   // ATAJ[3] := 3;
   // ATAJ[4] := 6;
   // ATAJ[5] := 5;
   // ATAB[1] := 1;
   // ATAB[2] := 2;
   // ATAB[3] := 3;
   // ATAB[4] := 4;
   // ATAB[5] := 5;
   // PSTT[1] := 1;
   // PSTT[2] := 2;
   // PSTT[3] := 3;
   // PSTT[4] := 4;
   // PSTT[5] := 5;
   // NSTT[0] := 1;
   // NSTT[1] := 2;
   // NSTT[2] := 3;
   // NSTT[3] := 4;
   // NSTT[4] := 5;
   // ASSJ[1] := 1;
   // ASSJ[2] := 2;
   // ASSJ[3] := 3;
   // ASSJ[4] := 4;
   // ASSJ[5] := 5;
   // ASSB[1] := 1;
   // ASSB[2] := 2;
   // ASSB[3] := 3;
   // ASSB[4] := 4;
   // ASSB[5] := 5;
   // PTTS[0] := 255;
   // PTTS[2] := 1;
   // PTTS[3] := 2;
   // PTTS[4] := 3;
   // PTTS[5] := 4;
   // NTTS[1] := 1;
   // NTTS[2] := 2;
   // NTTS[3] := 3;
   // NTTS[4] := 4;
   // NTTS[5] := 5;
   // TVX[0] := 16#1;
   // TTX[0] := 16#1;
   // TSX[0] := 16#1;
   // S00X[0] := 16#1;
   // SOFFX[0] := 16#1;
   // SONX[0] := 16#1;
   // SAX[0] := 16#1;
   // SERRX[0] := 16#1;
   // SMX[0] := 16#1;
   // S0X[0] := 16#1;
   // S1X[0] := 16#1;
   // LSTT[6] := 255;
   // ATAJ[6] := 4;
   // ATAB[0] := 6;
   // NSTT[6] := 5;
   // SW_SQTS[1] := 1;
   // SW_SQTS[2] := 1;
   // SW_SQTS[3] := 1;
   // SW_SQTS[4] := 1;
   // SW_SQTS[5] := 2;
BEGIN
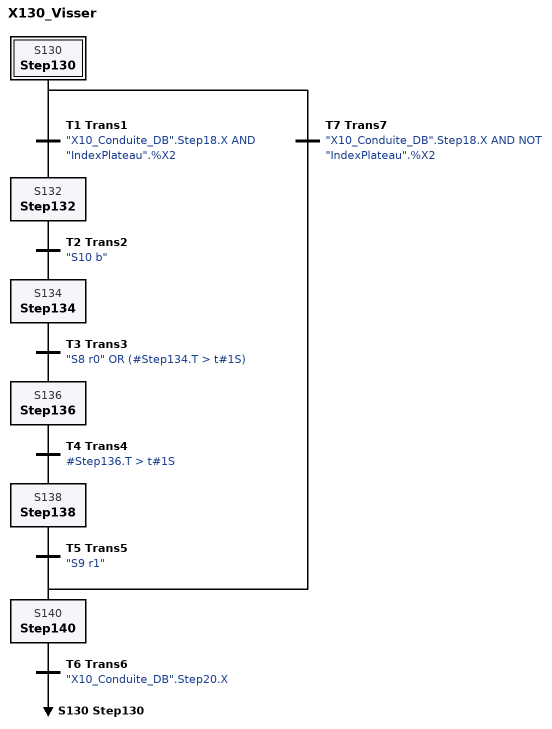
   // sequencer 1
   INITIAL_STEP Step130:   // S130, max time T#10S, warning time T#7S
   END_STEP
   TRANSITION Trans1 FROM Step130 TO Step132   // T1
      := "X10_Conduite_DB".Step18.X AND "IndexPlateau".%X2;
   END_TRANSITION
   TRANSITION Trans7 FROM Step130 TO Step140   // T7
      := "X10_Conduite_DB".Step18.X AND NOT "IndexPlateau".%X2;
   END_TRANSITION
   STEP Step132:   // S132, max time T#10S, warning time T#7S
   END_STEP
   TRANSITION Trans2 FROM Step132 TO Step134   // T2: Flacon bloqué
      := "S10 b";
   END_TRANSITION
   STEP Step134:   // S134, max time T#10S, warning time T#7S
   END_STEP
   TRANSITION Trans3 FROM Step134 TO Step136   // T3: Visseuse en bas
      := "S8 r0" OR (#Step134.T > t#1S);
   END_TRANSITION
   STEP Step136:   // S136, max time T#10S, warning time T#7S
   END_STEP
   TRANSITION Trans4 FROM Step136 TO Step138   // T4: Bouchon vissé
      := #Step136.T > t#1S;
   END_TRANSITION
   STEP Step138:   // S138, max time T#10S, warning time T#7S
   END_STEP
   TRANSITION Trans5 FROM Step138 TO Step140   // T5: Visseuse en haut
      := "S9 r1";
   END_TRANSITION
   STEP Step140:   // S140, max time T#10S, warning time T#7S
   END_STEP
   TRANSITION Trans6 FROM Step140 TO Step130   // T6, jump
      := "X10_Conduite_DB".Step20.X;
   END_TRANSITION
END_FUNCTION_BLOCK

FUNCTION_BLOCK "X160_Evacuer"   // FB5, GRAPH_PLUS
{ S7_Optimized_Access := 'TRUE' }
VERSION : 0.1
   VAR_INPUT
      OFF_SQ : Bool := false;   // Désactiver le graphe
      INIT_SQ : Bool := false;   // Mettre le graphe à l'état initial
      ACK_EF : Bool := false;   // Acquitter toutes les erreurs et perturbations
      S_PREV : Bool := false;   // Afficher l'étape précédente dans le paramètre S_NO
      S_NEXT : Bool := false;   // Afficher l'étape suivante dans le paramètre S_NO
      SW_AUTO : Bool := false;   // Mode automatique
      SW_TAP : Bool := false;   // Mode semi-automatique/Activation de l'étape suivante avec transition
      SW_TOP : Bool := false;   // Mode semi-automatique/Ignorer la transition
      SW_MAN : Bool := false;   // Mode manuel
      S_SEL : Int := 0;   // Sélectionner l'étape à afficher dans S_NO
      S_ON : Bool := false;   // Activer l'étape figurant dans le paramètre S_NO
      S_OFF : Bool := false;   // Désactiver l'étape figurant dans le paramètre S_NO
      T_PUSH : Bool := false;   // Validation de commutation pour transition en mode semi-automatique
   END_VAR
   VAR_OUTPUT
      S_NO : Int := 0;   // Numéro d'étape
      S_MORE : Bool := false;   // Il existe d'autres étapes qui peuvent être affichées dans S_NO.
      S_ACTIVE : Bool := false;   // L'étape affichée dans le paramètre S_NO est activée
      ERR_FLT : Bool := false;   // Erreur groupée Interlock or Supervision
      AUTO_ON : Bool := false;   // Mode automatique activé
      TAP_ON : Bool := false;   // Mode semi-automatique/Etape avec transition activé
      TOP_ON : Bool := false;   // Mode semi-automatique/Ignorer la transition activé
      MAN_ON : Bool := false;   // Mode manuel activé
   END_VAR
   VAR
      HMI_INFO : Array[0..8] of UInt;
      IF_PAR : G7_IfParPlus_V6;
      RT_DATA : G7_RTDataPlus_V6;   // Plage de données interne
      Trans1 : G7_TransitionPlus_V6;   // Structure de la transition
      Trans2 : G7_TransitionPlus_V6;   // Structure de la transition
      Trans3 : G7_TransitionPlus_V6;   // Structure de la transition
      Trans4 : G7_TransitionPlus_V6;   // Structure de la transition
      Step160 : G7_StepPlus_V6;   // Structure de l'étape
      Step162 : G7_StepPlus_V6;   // Structure de l'étape
      Step164 : G7_StepPlus_V6;   // Structure de l'étape
      SINI : Array[0..1] of USInt;
      LSTT : Array[0..3] of USInt;
      ATAJ : Array[0..3] of USInt;
      ATAB : Array[0..3] of USInt;
      PSTT : Array[0..3] of USInt;
      NSTT : Array[0..3] of USInt;
      ASSJ : Array[0..2] of USInt;
      ASSB : Array[0..2] of USInt;
      PTTS : Array[0..2] of USInt;
      NTTS : Array[0..2] of USInt;
      SW_SQTS : Array[0..2] of USInt;
      SWITCH : Array[0..1] of USInt;
      TVX : Array[0..3] of USInt;
      TTX : Array[0..3] of USInt;
      TSX : Array[0..1] of USInt;
      S00X : Array[0..1] of USInt;
      SOFFX : Array[0..1] of USInt;
      SONX : Array[0..1] of USInt;
      SAX : Array[0..1] of USInt;
      SERRX : Array[0..3] of USInt;
      SMX : Array[0..3] of USInt;
      S0X : Array[0..3] of USInt;
      S1X : Array[0..3] of USInt;
      IL_ALARM_INST : Diag_Alarm;
      SUP_ALARM_INST : Diag_Alarm;
      STEP_TIME_ALARM_INST : Diag_Alarm;
      IEC_TIMER_INST : IEC_TIMER;
      TRANSACTION_FLAG : Bool := false;
   END_VAR
   // SINI[0] := 2;
   // LSTT[0] := 255;
   // LSTT[1] := 255;
   // ATAJ[1] := 3;
   // ATAJ[2] := 2;
   // ATAB[1] := 1;
   // ATAB[2] := 2;
   // PSTT[1] := 1;
   // PSTT[2] := 2;
   // NSTT[0] := 1;
   // NSTT[1] := 2;
   // ASSJ[1] := 1;
   // ASSJ[2] := 2;
   // ASSB[1] := 1;
   // ASSB[2] := 2;
   // PTTS[0] := 255;
   // PTTS[2] := 1;
   // NTTS[1] := 1;
   // NTTS[2] := 2;
   // TVX[0] := 16#1;
   // TTX[0] := 16#1;
   // TSX[0] := 16#1;
   // S00X[0] := 16#1;
   // SOFFX[0] := 16#1;
   // SONX[0] := 16#1;
   // SAX[0] := 16#1;
   // SERRX[0] := 16#1;
   // SMX[0] := 16#1;
   // S0X[0] := 16#1;
   // S1X[0] := 16#1;
   // LSTT[3] := 255;
   // ATAJ[3] := 1;
   // ATAB[0] := 3;
   // NSTT[3] := 2;
   // SW_SQTS[1] := 1;
   // SW_SQTS[2] := 2;
BEGIN
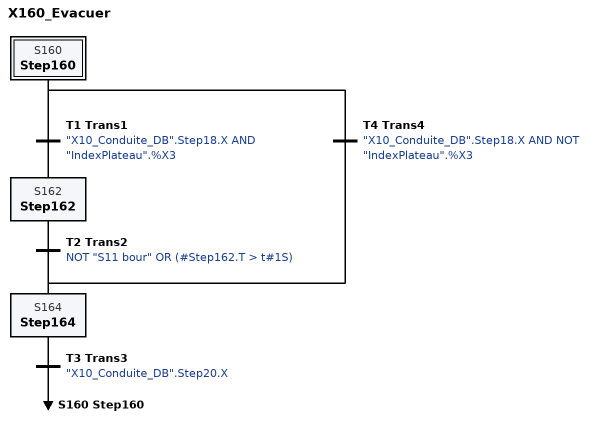
   // sequencer 1
   INITIAL_STEP Step160:   // S160, max time T#10S, warning time T#7S
   END_STEP
   TRANSITION Trans1 FROM Step160 TO Step162   // T1
      := "X10_Conduite_DB".Step18.X AND "IndexPlateau".%X3;
   END_TRANSITION
   TRANSITION Trans4 FROM Step160 TO Step164   // T4
      := "X10_Conduite_DB".Step18.X AND NOT "IndexPlateau".%X3;
   END_TRANSITION
   STEP Step162:   // S162, max time T#10S, warning time T#7S
   END_STEP
   TRANSITION Trans2 FROM Step162 TO Step164   // T2: Flacon évacué
      := NOT "S11 bour" OR (#Step162.T > t#1S);
   END_TRANSITION
   STEP Step164:   // S164, max time T#10S, warning time T#7S
   END_STEP
   TRANSITION Trans3 FROM Step164 TO Step160   // T3, jump
      := "X10_Conduite_DB".Step20.X;
   END_TRANSITION
END_FUNCTION_BLOCK

FUNCTION_BLOCK "X10_Conduite"   // FB6, GRAPH_PLUS
{ S7_Optimized_Access := 'TRUE' }
VERSION : 0.1
   VAR_INPUT
      OFF_SQ : Bool := false;   // Désactiver le graphe
      INIT_SQ : Bool := false;   // Mettre le graphe à l'état initial
      ACK_EF : Bool := false;   // Acquitter toutes les erreurs et perturbations
      S_PREV : Bool := false;   // Afficher l'étape précédente dans le paramètre S_NO
      S_NEXT : Bool := false;   // Afficher l'étape suivante dans le paramètre S_NO
      SW_AUTO : Bool := false;   // Mode automatique
      SW_TAP : Bool := false;   // Mode semi-automatique/Activation de l'étape suivante avec transition
      SW_TOP : Bool := false;   // Mode semi-automatique/Ignorer la transition
      SW_MAN : Bool := false;   // Mode manuel
      S_SEL : Int := 0;   // Sélectionner l'étape à afficher dans S_NO
      S_ON : Bool := false;   // Activer l'étape figurant dans le paramètre S_NO
      S_OFF : Bool := false;   // Désactiver l'étape figurant dans le paramètre S_NO
      T_PUSH : Bool := false;   // Validation de commutation pour transition en mode semi-automatique
   END_VAR
   VAR_OUTPUT
      S_NO : Int := 0;   // Numéro d'étape
      S_MORE : Bool := false;   // Il existe d'autres étapes qui peuvent être affichées dans S_NO.
      S_ACTIVE : Bool := false;   // L'étape affichée dans le paramètre S_NO est activée
      ERR_FLT : Bool := false;   // Erreur groupée Interlock or Supervision
      AUTO_ON : Bool := false;   // Mode automatique activé
      TAP_ON : Bool := false;   // Mode semi-automatique/Etape avec transition activé
      TOP_ON : Bool := false;   // Mode semi-automatique/Ignorer la transition activé
      MAN_ON : Bool := false;   // Mode manuel activé
   END_VAR
   VAR
      HMI_INFO : Array[0..8] of UInt;
      IF_PAR : G7_IfParPlus_V6;
      RT_DATA : G7_RTDataPlus_V6;   // Plage de données interne
      Trans1 : G7_TransitionPlus_V6;   // Structure de la transition
      Trans2 : G7_TransitionPlus_V6;   // Structure de la transition
      Trans3 : G7_TransitionPlus_V6;   // Structure de la transition
      Trans4 : G7_TransitionPlus_V6;   // Structure de la transition
      Trans5 : G7_TransitionPlus_V6;   // Structure de la transition
      Trans6 : G7_TransitionPlus_V6;   // Structure de la transition
      Trans8 : G7_TransitionPlus_V6;   // Structure de la transition
      Trans9 : G7_TransitionPlus_V6;   // Structure de la transition
      Trans10 : G7_TransitionPlus_V6;   // Structure de la transition
      Trans11 : G7_TransitionPlus_V6;   // Structure de la transition
      Trans13 : G7_TransitionPlus_V6;   // Structure de la transition
      Trans15 : G7_TransitionPlus_V6;   // Structure de la transition
      Trans16 : G7_TransitionPlus_V6;   // Structure de la transition
      Trans17 : G7_TransitionPlus_V6;   // Structure de la transition
      Step10 : G7_StepPlus_V6;   // Structure de l'étape
      Step12 : G7_StepPlus_V6;   // Structure de l'étape
      Step13 : G7_StepPlus_V6;   // Structure de l'étape
      Step14 : G7_StepPlus_V6;   // Structure de l'étape
      Step15 : G7_StepPlus_V6;   // Structure de l'étape
      Step16 : G7_StepPlus_V6;   // Structure de l'étape
      Step18 : G7_StepPlus_V6;   // Structure de l'étape
      Step20 : G7_StepPlus_V6;   // Structure de l'étape
      SINI : Array[0..1] of USInt;
      LSTT : Array[0..13] of USInt;
      ATAJ : Array[0..13] of USInt;
      ATAB : Array[0..13] of USInt;
      PSTT : Array[0..13] of USInt;
      NSTT : Array[0..13] of USInt;
      ASSJ : Array[0..7] of USInt;
      ASSB : Array[0..7] of USInt;
      PTTS : Array[0..7] of USInt;
      NTTS : Array[0..7] of USInt;
      SW_SQTS : Array[0..7] of USInt;
      SWITCH : Array[0..4] of USInt;
      TVX : Array[0..12] of USInt;
      TTX : Array[0..12] of USInt;
      TSX : Array[0..1] of USInt;
      S00X : Array[0..1] of USInt;
      SOFFX : Array[0..1] of USInt;
      SONX : Array[0..1] of USInt;
      SAX : Array[0..1] of USInt;
      SERRX : Array[0..8] of USInt;
      SMX : Array[0..8] of USInt;
      S0X : Array[0..8] of USInt;
      S1X : Array[0..8] of USInt;
      IL_ALARM_INST : Diag_Alarm;
      SUP_ALARM_INST : Diag_Alarm;
      STEP_TIME_ALARM_INST : Diag_Alarm;
      IEC_TIMER_INST : IEC_TIMER;
      TRANSACTION_FLAG : Bool := false;
   END_VAR
   // SINI[0] := 2;
   // LSTT[0] := 255;
   // LSTT[1] := 255;
   // LSTT[2] := 255;
   // LSTT[3] := 255;
   // LSTT[4] := 255;
   // LSTT[6] := 255;
   // ATAJ[1] := 8;
   // ATAJ[2] := 2;
   // ATAJ[3] := 3;
   // ATAJ[4] := 4;
   // ATAJ[5] := 5;
   // ATAJ[6] := 6;
   // ATAB[1] := 9;
   // ATAB[2] := 10;
   // ATAB[3] := 11;
   // ATAB[4] := 12;
   // ATAB[5] := 5;
   // ATAB[6] := 6;
   // PSTT[1] := 1;
   // PSTT[2] := 3;
   // PSTT[3] := 5;
   // PSTT[4] := 6;
   // PSTT[5] := 7;
   // PSTT[6] := 2;
   // NSTT[0] := 1;
   // NSTT[1] := 2;
   // NSTT[2] := 5;
   // NSTT[3] := 6;
   // NSTT[4] := 7;
   // NSTT[6] := 3;
   // ASSJ[1] := 1;
   // ASSJ[2] := 2;
   // ASSJ[3] := 3;
   // ASSJ[4] := 4;
   // ASSJ[5] := 5;
   // ASSJ[6] := 6;
   // ASSB[1] := 1;
   // ASSB[2] := 2;
   // ASSB[3] := 3;
   // ASSB[4] := 4;
   // ASSB[5] := 5;
   // ASSB[6] := 6;
   // PTTS[0] := 255;
   // PTTS[2] := 1;
   // PTTS[3] := 6;
   // PTTS[4] := 7;
   // PTTS[5] := 2;
   // PTTS[6] := 3;
   // NTTS[1] := 1;
   // NTTS[2] := 6;
   // NTTS[3] := 2;
   // NTTS[4] := 8;
   // NTTS[5] := 3;
   // NTTS[6] := 4;
   // TVX[0] := 16#1;
   // TTX[0] := 16#1;
   // TSX[0] := 16#1;
   // S00X[0] := 16#1;
   // SOFFX[0] := 16#1;
   // SONX[0] := 16#1;
   // SAX[0] := 16#1;
   // SERRX[0] := 16#1;
   // SMX[0] := 16#1;
   // S0X[0] := 16#1;
   // S1X[0] := 16#1;
   // LSTT[7] := 255;
   // LSTT[8] := 255;
   // ATAJ[7] := 7;
   // ATAJ[8] := 1;
   // ATAB[7] := 1;
   // ATAB[8] := 13;
   // PSTT[7] := 1;
   // PSTT[8] := 4;
   // NSTT[7] := 4;
   // NSTT[8] := 2;
   // ASSJ[7] := 7;
   // ASSB[7] := 7;
   // PTTS[7] := 4;
   // NTTS[7] := 5;
   // SW_SQTS[2] := 1;
   // SW_SQTS[3] := 1;
   // SW_SQTS[4] := 2;
   // SW_SQTS[5] := 3;
   // SW_SQTS[6] := 4;
   // SW_SQTS[7] := 5;
   // ATAJ[9] := 9;
   // ATAJ[10] := 10;
   // ATAJ[11] := 11;
   // ATAJ[12] := 12;
   // ATAB[9] := 7;
   // ATAB[10] := 2;
   // ATAB[11] := 3;
   // ATAB[12] := 4;
   // PSTT[9] := 1;
   // PSTT[10] := 3;
   // PSTT[11] := 5;
   // PSTT[12] := 6;
   // ATAJ[13] := 13;
   // ATAB[13] := 8;
   // PSTT[13] := 4;
BEGIN
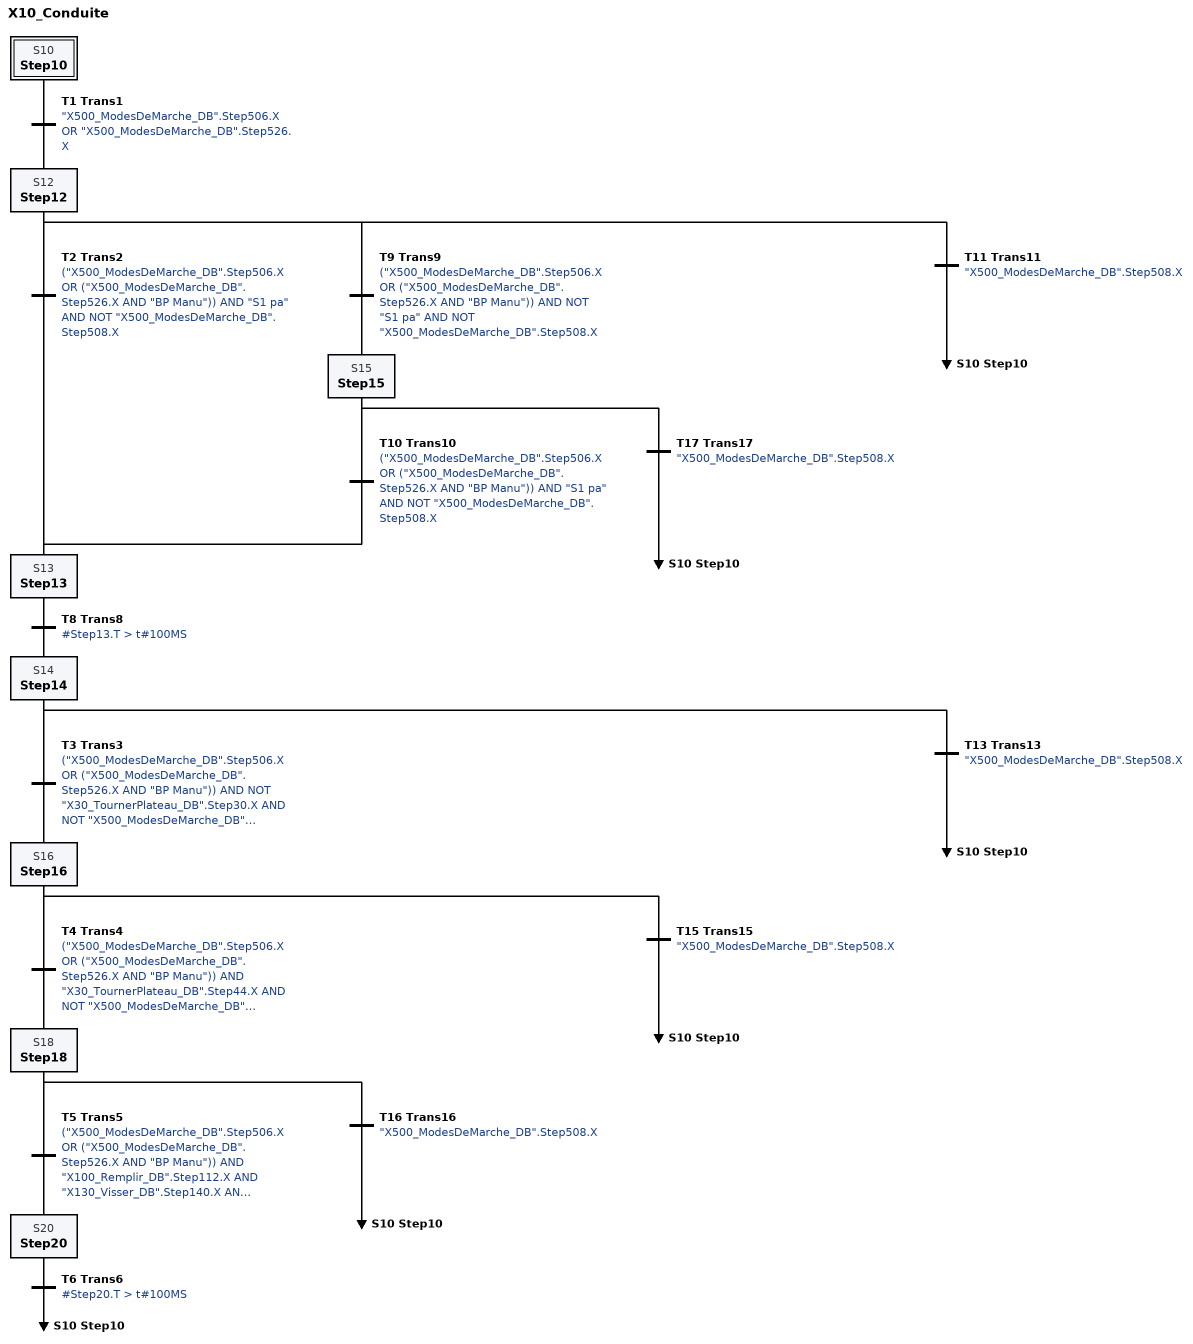
   // sequencer 1
   INITIAL_STEP Step10:   // S10, max time T#10S, warning time T#7S
   END_STEP
   TRANSITION Trans1 FROM Step10 TO Step12   // T1: Cycle auto ou manu en cours
      := "X500_ModesDeMarche_DB".Step506.X OR "X500_ModesDeMarche_DB".Step526.X;
   END_TRANSITION
   STEP Step12:   // S12, max time T#10S, warning time T#7S
   END_STEP
   TRANSITION Trans2 FROM Step12 TO Step13   // T2: Flacons présents en entrée
      := ("X500_ModesDeMarche_DB".Step506.X OR ("X500_ModesDeMarche_DB".Step526.X AND "BP Manu")) AND "S1 pa" AND NOT "X500_ModesDeMarche_DB".Step508.X;
   END_TRANSITION
   TRANSITION Trans9 FROM Step12 TO Step15   // T9: Pas de flacon en entree
      := ("X500_ModesDeMarche_DB".Step506.X OR ("X500_ModesDeMarche_DB".Step526.X AND "BP Manu")) AND NOT "S1 pa" AND NOT "X500_ModesDeMarche_DB".Step508.X;
   END_TRANSITION
   TRANSITION Trans11 FROM Step12 TO Step10   // T11, jump: Defaut present
      := "X500_ModesDeMarche_DB".Step508.X;
   END_TRANSITION
   STEP Step14:   // S14, max time T#10S, warning time T#7S
   END_STEP
   TRANSITION Trans3 FROM Step14 TO Step16   // T3: Tourner plateau en cours
      := ("X500_ModesDeMarche_DB".Step506.X OR ("X500_ModesDeMarche_DB".Step526.X AND "BP Manu")) AND NOT "X30_TournerPlateau_DB".Step30.X AND NOT "X500_ModesDeMarche_DB".Step508.X;
   END_TRANSITION
   TRANSITION Trans13 FROM Step14 TO Step10   // T13, jump: Defaut present
      := "X500_ModesDeMarche_DB".Step508.X;
   END_TRANSITION
   STEP Step16:   // S16, max time T#10S, warning time T#7S
   END_STEP
   TRANSITION Trans4 FROM Step16 TO Step18   // T4: Fin de tourner plateau
      := ("X500_ModesDeMarche_DB".Step506.X OR ("X500_ModesDeMarche_DB".Step526.X AND "BP Manu")) AND "X30_TournerPlateau_DB".Step44.X AND NOT "X500_ModesDeMarche_DB".Step508.X AND (#Step16.T > t#100MS);
   END_TRANSITION
   TRANSITION Trans15 FROM Step16 TO Step10   // T15, jump: Defaut present
      := "X500_ModesDeMarche_DB".Step508.X;
   END_TRANSITION
   STEP Step18:   // S18, max time T#10S, warning time T#7S
   END_STEP
   TRANSITION Trans5 FROM Step18 TO Step20   // T5: Pilotage terminés
      := ("X500_ModesDeMarche_DB".Step506.X OR ("X500_ModesDeMarche_DB".Step526.X AND "BP Manu")) AND "X100_Remplir_DB".Step112.X AND "X130_Visser_DB".Step140.X AND "X160_Evacuer_DB".Step164.X AND NOT "X500_ModesDeMarche_DB".Step508.X;
   END_TRANSITION
   TRANSITION Trans16 FROM Step18 TO Step10   // T16, jump: Defaut present
      := "X500_ModesDeMarche_DB".Step508.X;
   END_TRANSITION
   STEP Step20:   // S20, max time T#10S, warning time T#7S
   END_STEP
   TRANSITION Trans6 FROM Step20 TO Step10   // T6, jump: Fin
      := #Step20.T > t#100MS;
   END_TRANSITION
   STEP Step13:   // S13, max time T#10S, warning time T#7S
   END_STEP
   TRANSITION Trans8 FROM Step13 TO Step14   // T8: Latence pour incrementation index
      := #Step13.T > t#100MS;
   END_TRANSITION
   STEP Step15:   // S15, max time T#10S, warning time T#7S
   END_STEP
   TRANSITION Trans10 FROM Step15 TO Step13   // T10: Flacon en entrée
      := ("X500_ModesDeMarche_DB".Step506.X OR ("X500_ModesDeMarche_DB".Step526.X AND "BP Manu")) AND "S1 pa" AND NOT "X500_ModesDeMarche_DB".Step508.X;
   END_TRANSITION
   TRANSITION Trans17 FROM Step15 TO Step10   // T17, jump: Defaut
      := "X500_ModesDeMarche_DB".Step508.X;
   END_TRANSITION
END_FUNCTION_BLOCK

FUNCTION_BLOCK "GestionIndexPlateau"   // FB7, LAD
{ S7_Optimized_Access := 'TRUE' }
VERSION : 0.1
   VAR
      FM1 : Bool;
   END_VAR
   VAR_TEMP   // added for the SCL form of the ladder/FBD networks
      _w1 : Bool;
   END_VAR
BEGIN

REGION Network 1: Décalage de l'index si plateau tourne
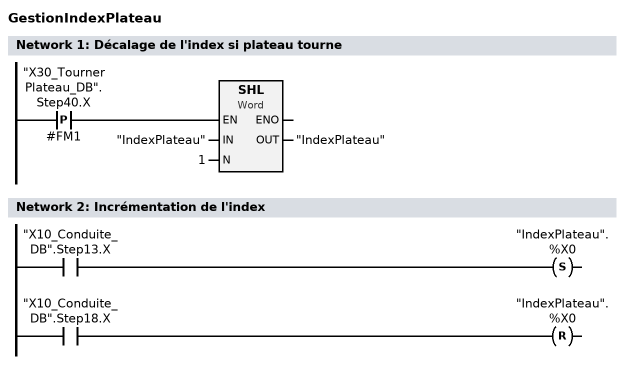
   RUNG wire#powerrail
      P_Contact(operand := "X30_TournerPlateau_DB".Step40.X, bit := #FM1)
      { S7_Templates := "SrcType := Word" } Shl(in := "IndexPlateau", n := 1, out => "IndexPlateau")
   END_RUNG
   // the same network as SCL:
   #_w1 := "X30_TournerPlateau_DB".Step40.X AND NOT #FM1;   // rising edge of "X30_TournerPlateau_DB".Step40.X
   #FM1 := "X30_TournerPlateau_DB".Step40.X;
   IF #_w1 THEN "IndexPlateau" := SHL(IN := "IndexPlateau", N := 1); END_IF;
END_REGION

REGION Network 2: Incrémentation de l'index
   RUNG wire#powerrail
      Contact( "X10_Conduite_DB".Step13.X )
      S_Coil( "IndexPlateau".%X0 )
   END_RUNG
   RUNG wire#powerrail
      Contact( "X10_Conduite_DB".Step18.X )
      R_Coil( "IndexPlateau".%X0 )
   END_RUNG
   // the same network as SCL:
   IF "X10_Conduite_DB".Step13.X THEN "IndexPlateau".%X0 := TRUE; END_IF;
   IF "X10_Conduite_DB".Step18.X THEN "IndexPlateau".%X0 := FALSE; END_IF;
END_REGION
END_FUNCTION_BLOCK

FUNCTION_BLOCK "X500_ModesDeMarche"   // FB8, GRAPH_PLUS
{ S7_Optimized_Access := 'TRUE' }
VERSION : 0.1
   VAR_INPUT
      OFF_SQ : Bool := false;   // Désactiver le graphe
      INIT_SQ : Bool := false;   // Mettre le graphe à l'état initial
      ACK_EF : Bool := false;   // Acquitter toutes les erreurs et perturbations
      S_PREV : Bool := false;   // Afficher l'étape précédente dans le paramètre S_NO
      S_NEXT : Bool := false;   // Afficher l'étape suivante dans le paramètre S_NO
      SW_AUTO : Bool := false;   // Mode automatique
      SW_TAP : Bool := false;   // Mode semi-automatique/Activation de l'étape suivante avec transition
      SW_TOP : Bool := false;   // Mode semi-automatique/Ignorer la transition
      SW_MAN : Bool := false;   // Mode manuel
      S_SEL : Int := 0;   // Sélectionner l'étape à afficher dans S_NO
      S_ON : Bool := false;   // Activer l'étape figurant dans le paramètre S_NO
      S_OFF : Bool := false;   // Désactiver l'étape figurant dans le paramètre S_NO
      T_PUSH : Bool := false;   // Validation de commutation pour transition en mode semi-automatique
   END_VAR
   VAR_OUTPUT
      S_NO : Int := 0;   // Numéro d'étape
      S_MORE : Bool := false;   // Il existe d'autres étapes qui peuvent être affichées dans S_NO.
      S_ACTIVE : Bool := false;   // L'étape affichée dans le paramètre S_NO est activée
      ERR_FLT : Bool := false;   // Erreur groupée Interlock or Supervision
      AUTO_ON : Bool := false;   // Mode automatique activé
      TAP_ON : Bool := false;   // Mode semi-automatique/Etape avec transition activé
      TOP_ON : Bool := false;   // Mode semi-automatique/Ignorer la transition activé
      MAN_ON : Bool := false;   // Mode manuel activé
   END_VAR
   VAR
      HMI_INFO : Array[0..8] of UInt;
      IF_PAR : G7_IfParPlus_V6;
      RT_DATA : G7_RTDataPlus_V6;   // Plage de données interne
      Trans1 : G7_TransitionPlus_V6;   // Structure de la transition
      Trans2 : G7_TransitionPlus_V6;   // Structure de la transition
      Trans3 : G7_TransitionPlus_V6;   // Structure de la transition
      Trans4 : G7_TransitionPlus_V6;   // Structure de la transition
      Trans5 : G7_TransitionPlus_V6;   // Structure de la transition
      Trans6 : G7_TransitionPlus_V6;   // Structure de la transition
      Trans7 : G7_TransitionPlus_V6;   // Structure de la transition
      Trans8 : G7_TransitionPlus_V6;   // Structure de la transition
      Trans9 : G7_TransitionPlus_V6;   // Structure de la transition
      Trans10 : G7_TransitionPlus_V6;   // Structure de la transition
      Trans11 : G7_TransitionPlus_V6;   // Structure de la transition
      Trans12 : G7_TransitionPlus_V6;   // Structure de la transition
      Trans13 : G7_TransitionPlus_V6;   // Structure de la transition
      Trans14 : G7_TransitionPlus_V6;   // Structure de la transition
      Trans15 : G7_TransitionPlus_V6;   // Structure de la transition
      Trans16 : G7_TransitionPlus_V6;   // Structure de la transition
      Step500 : G7_StepPlus_V6;   // Structure de l'étape
      Step502 : G7_StepPlus_V6;   // Structure de l'étape
      Step504 : G7_StepPlus_V6;   // Structure de l'étape
      Step506 : G7_StepPlus_V6;   // Structure de l'étape
      Step508 : G7_StepPlus_V6;   // Structure de l'étape
      Step524 : G7_StepPlus_V6;   // Structure de l'étape
      Step526 : G7_StepPlus_V6;   // Structure de l'étape
      Step528 : G7_StepPlus_V6;   // Structure de l'étape
      Step542 : G7_StepPlus_V6;   // Structure de l'étape
      SINI : Array[0..1] of USInt;
      LSTT : Array[0..15] of USInt;
      ATAJ : Array[0..15] of USInt;
      ATAB : Array[0..15] of USInt;
      PSTT : Array[0..15] of USInt;
      NSTT : Array[0..15] of USInt;
      ASSJ : Array[0..8] of USInt;
      ASSB : Array[0..8] of USInt;
      PTTS : Array[0..8] of USInt;
      NTTS : Array[0..8] of USInt;
      SW_SQTS : Array[0..8] of USInt;
      SWITCH : Array[0..10] of USInt;
      TVX : Array[0..14] of USInt;
      TTX : Array[0..14] of USInt;
      TSX : Array[0..1] of USInt;
      S00X : Array[0..1] of USInt;
      SOFFX : Array[0..1] of USInt;
      SONX : Array[0..1] of USInt;
      SAX : Array[0..1] of USInt;
      SERRX : Array[0..9] of USInt;
      SMX : Array[0..9] of USInt;
      S0X : Array[0..9] of USInt;
      S1X : Array[0..9] of USInt;
      IL_ALARM_INST : Diag_Alarm;
      SUP_ALARM_INST : Diag_Alarm;
      STEP_TIME_ALARM_INST : Diag_Alarm;
      IEC_TIMER_INST : IEC_TIMER;
      TRANSACTION_FLAG : Bool := false;
   END_VAR
   // SINI[0] := 2;
   // LSTT[0] := 255;
   // LSTT[1] := 255;
   // LSTT[2] := 1;
   // LSTT[3] := 255;
   // LSTT[4] := 255;
   // LSTT[5] := 1;
   // LSTT[6] := 255;
   // LSTT[7] := 255;
   // LSTT[9] := 255;
   // LSTT[10] := 2;
   // LSTT[11] := 1;
   // LSTT[13] := 255;
   // LSTT[14] := 5;
   // ATAJ[1] := 1;
   // ATAJ[2] := 2;
   // ATAJ[3] := 3;
   // ATAJ[4] := 4;
   // ATAJ[5] := 5;
   // ATAJ[6] := 6;
   // ATAJ[7] := 7;
   // ATAJ[8] := 8;
   // ATAJ[9] := 9;
   // ATAJ[10] := 10;
   // ATAJ[11] := 11;
   // ATAJ[12] := 12;
   // ATAJ[13] := 13;
   // ATAJ[14] := 14;
   // ATAB[0] := 1;
   // ATAB[2] := 2;
   // ATAB[3] := 15;
   // ATAB[4] := 3;
   // ATAB[5] := 7;
   // ATAB[6] := 11;
   // ATAB[7] := 5;
   // ATAB[8] := 9;
   // ATAB[9] := 8;
   // ATAB[10] := 10;
   // ATAB[11] := 6;
   // ATAB[12] := 13;
   // ATAB[13] := 12;
   // ATAB[14] := 14;
   // PSTT[2] := 8;
   // PSTT[3] := 1;
   // PSTT[4] := 1;
   // PSTT[5] := 2;
   // PSTT[6] := 5;
   // PSTT[7] := 2;
   // PSTT[8] := 3;
   // PSTT[9] := 3;
   // PSTT[10] := 4;
   // PSTT[11] := 5;
   // PSTT[12] := 6;
   // PSTT[13] := 6;
   // PSTT[14] := 7;
   // NSTT[0] := 1;
   // NSTT[1] := 8;
   // NSTT[2] := 1;
   // NSTT[3] := 2;
   // NSTT[4] := 5;
   // NSTT[5] := 1;
   // NSTT[6] := 6;
   // NSTT[7] := 3;
   // NSTT[9] := 4;
   // NSTT[10] := 2;
   // NSTT[11] := 1;
   // NSTT[13] := 7;
   // NSTT[14] := 5;
   // ASSJ[1] := 1;
   // ASSJ[2] := 2;
   // ASSJ[3] := 3;
   // ASSJ[4] := 4;
   // ASSJ[5] := 5;
   // ASSJ[6] := 6;
   // ASSJ[7] := 7;
   // ASSJ[8] := 8;
   // ASSB[1] := 1;
   // ASSB[2] := 2;
   // ASSB[3] := 3;
   // ASSB[4] := 4;
   // ASSB[5] := 5;
   // ASSB[6] := 6;
   // ASSB[7] := 7;
   // ASSB[8] := 8;
   // PTTS[0] := 255;
   // PTTS[2] := 3;
   // PTTS[3] := 7;
   // PTTS[4] := 9;
   // PTTS[5] := 4;
   // PTTS[6] := 6;
   // PTTS[7] := 13;
   // PTTS[8] := 1;
   // NTTS[1] := 3;
   // NTTS[2] := 5;
   // NTTS[3] := 8;
   // NTTS[4] := 10;
   // NTTS[5] := 6;
   // NTTS[6] := 12;
   // NTTS[7] := 14;
   // NTTS[8] := 2;
   // SW_SQTS[1] := 1;
   // SW_SQTS[2] := 2;
   // SW_SQTS[3] := 3;
   // SW_SQTS[4] := 4;
   // SW_SQTS[5] := 5;
   // SW_SQTS[6] := 6;
   // SW_SQTS[7] := 7;
   // SW_SQTS[8] := 8;
   // TVX[0] := 16#1;
   // TTX[0] := 16#1;
   // TSX[0] := 16#1;
   // S00X[0] := 16#1;
   // SOFFX[0] := 16#1;
   // SONX[0] := 16#1;
   // SAX[0] := 16#1;
   // SERRX[0] := 16#1;
   // SMX[0] := 16#1;
   // S0X[0] := 16#1;
   // S1X[0] := 16#1;
   // ATAJ[15] := 15;
   // ATAB[15] := 4;
   // PSTT[15] := 1;
BEGIN
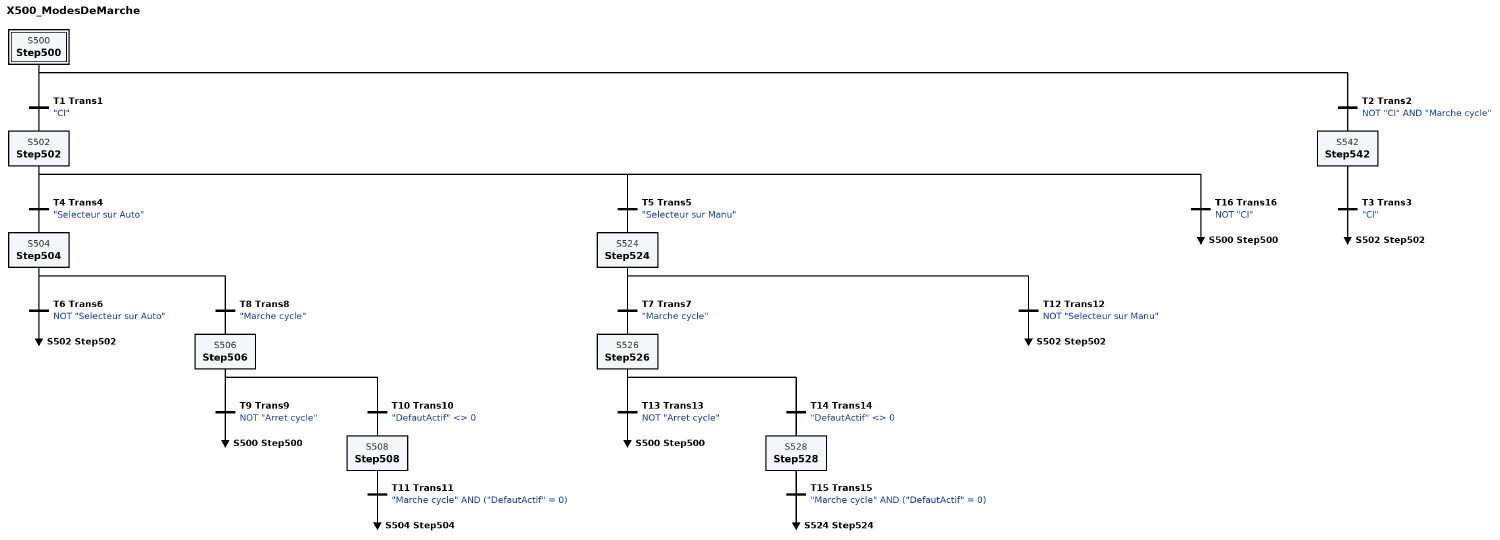
   // sequencer 1
   INITIAL_STEP Step500:   // S500, max time T#10S, warning time T#7S
   END_STEP
   TRANSITION Trans1 FROM Step500 TO Step502   // T1: Conditions initiales
      := "CI";
   END_TRANSITION
   TRANSITION Trans2 FROM Step500 TO Step542   // T2: Pas les conditions initiales
      := NOT "CI" AND "Marche cycle";
   END_TRANSITION
   STEP Step542:   // S542, max time T#10S, warning time T#7S
   END_STEP
   TRANSITION Trans3 FROM Step542 TO Step502   // T3, jump
      := "CI";
   END_TRANSITION
   STEP Step502:   // S502, max time T#10S, warning time T#7S
   END_STEP
   TRANSITION Trans4 FROM Step502 TO Step504   // T4: Selection Auto
      := "Selecteur sur Auto";
   END_TRANSITION
   TRANSITION Trans5 FROM Step502 TO Step524   // T5: Selection Manu
      := "Selecteur sur Manu";
   END_TRANSITION
   TRANSITION Trans16 FROM Step502 TO Step500   // T16, jump: Perte des CI
      := NOT "CI";
   END_TRANSITION
   STEP Step504:   // S504, max time T#10S, warning time T#7S
   END_STEP
   TRANSITION Trans6 FROM Step504 TO Step502   // T6, jump: Perte Select Auto
      := NOT "Selecteur sur Auto";
   END_TRANSITION
   TRANSITION Trans8 FROM Step504 TO Step506   // T8: Depart cycle
      := "Marche cycle";
   END_TRANSITION
   STEP Step524:   // S524, max time T#10S, warning time T#7S
   END_STEP
   TRANSITION Trans7 FROM Step524 TO Step526   // T7: Depart cycle
      := "Marche cycle";
   END_TRANSITION
   TRANSITION Trans12 FROM Step524 TO Step502   // T12, jump: Perte Select Manu
      := NOT "Selecteur sur Manu";
   END_TRANSITION
   STEP Step506:   // S506, max time T#10S, warning time T#7S
   END_STEP
   TRANSITION Trans9 FROM Step506 TO Step500   // T9, jump: Arret Cycle
      := NOT "Arret cycle";
   END_TRANSITION
   TRANSITION Trans10 FROM Step506 TO Step508   // T10: Defaut present
      := "DefautActif" <> 0;
   END_TRANSITION
   STEP Step508:   // S508, max time T#10S, warning time T#7S
   END_STEP
   TRANSITION Trans11 FROM Step508 TO Step504   // T11, jump: Pas de defaut et dcy
      := "Marche cycle" AND ("DefautActif" = 0);
   END_TRANSITION
   STEP Step526:   // S526, max time T#10S, warning time T#7S
   END_STEP
   TRANSITION Trans13 FROM Step526 TO Step500   // T13, jump: Arret cycle
      := NOT "Arret cycle";
   END_TRANSITION
   TRANSITION Trans14 FROM Step526 TO Step528   // T14: Defaut present
      := "DefautActif" <> 0;
   END_TRANSITION
   STEP Step528:   // S528, max time T#10S, warning time T#7S
   END_STEP
   TRANSITION Trans15 FROM Step528 TO Step524   // T15, jump: Pas de defaut et dcy
      := "Marche cycle" AND ("DefautActif" = 0);
   END_TRANSITION
END_FUNCTION_BLOCK

FUNCTION_BLOCK "CondInitiales"   // FB9, LAD
{ S7_Optimized_Access := 'TRUE' }
VERSION : 0.1
BEGIN

REGION Network 1: Condition initiales ok
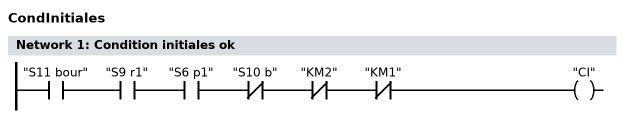
   RUNG wire#powerrail
      Contact( "S11 bour" )
      Contact( "S9 r1" )
      Contact( "S6 p1" )
      I_Contact( "S10 b" )
      I_Contact( "KM2" )
      I_Contact( "KM1" )
      Coil( "CI" )
   END_RUNG
   // the same network as SCL:
   "CI" := "S11 bour" AND "S9 r1" AND "S6 p1" AND NOT "S10 b" AND NOT "KM2" AND NOT "KM1";
END_REGION
END_FUNCTION_BLOCK

FUNCTION_BLOCK "defauts"   // FB10, LAD
{ S7_Optimized_Access := 'TRUE' }
VERSION : 0.1
BEGIN

REGION Network 1: Défaut actif : X0 = Pas de flacons en entrée
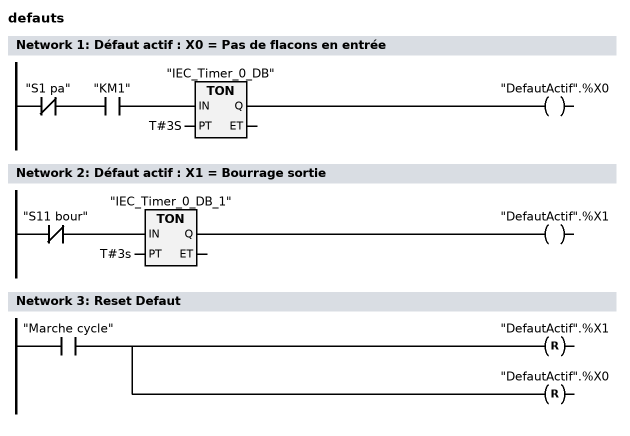
   "IEC_Timer_0_DB".TON(IN := NOT "S1 pa" AND "KM1", PT := T#3S);
   "DefautActif".%X0 := "IEC_Timer_0_DB".Q;
END_REGION

REGION Network 2: Défaut actif : X1 = Bourrage sortie
   "IEC_Timer_0_DB_1".TON(IN := NOT "S11 bour", PT := T#3s);
   "DefautActif".%X1 := "IEC_Timer_0_DB_1".Q;
END_REGION

REGION Network 3: Reset Defaut
   RUNG wire#powerrail
      Contact( "Marche cycle" )
      wire#w1
      R_Coil( "DefautActif".%X1 )
   END_RUNG
   RUNG wire#w1
      R_Coil( "DefautActif".%X0 )
   END_RUNG
   // the same network as SCL:
   IF "Marche cycle" THEN
       "DefautActif".%X1 := FALSE;
       "DefautActif".%X0 := FALSE;
   END_IF;
END_REGION
END_FUNCTION_BLOCK

ORGANIZATION_BLOCK "Main"   // OB1, LAD, ProgramCycle
TITLE = "Main Program Sweep (Cycle)"
{ S7_Optimized_Access := 'TRUE' }
VERSION : 0.1
   VAR_INPUT
      Initial_Call : Bool;   // Initial call of this OB
      Remanence : Bool;   // =True, if remanent data are available
   END_VAR
BEGIN

REGION Network 1: X30 : Tourner le plateau
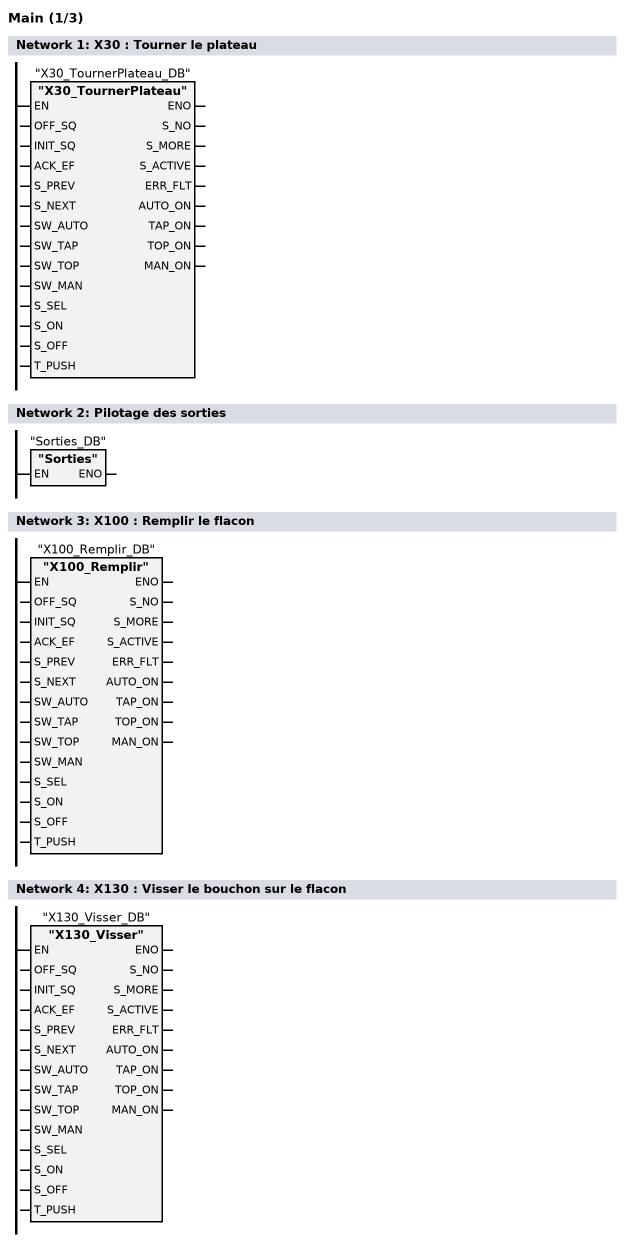
   RUNG wire#powerrail
      "X30_TournerPlateau_DB"(OFF_SQ :=, INIT_SQ :=, ACK_EF :=, S_PREV :=, S_NEXT :=, SW_AUTO :=, SW_TAP :=, SW_TOP :=, SW_MAN :=, S_SEL :=, S_ON :=, S_OFF :=, T_PUSH :=, S_NO =>, S_MORE =>, S_ACTIVE =>, ERR_FLT =>, AUTO_ON =>, TAP_ON =>, TOP_ON =>, MAN_ON =>)
   END_RUNG
   // the same network as SCL:
   "X30_TournerPlateau_DB"();   // "X30_TournerPlateau"
END_REGION

REGION Network 2: Pilotage des sorties
   RUNG wire#powerrail
      "Sorties_DB"()
   END_RUNG
   // the same network as SCL:
   "Sorties_DB"();   // "Sorties"
END_REGION

REGION Network 3: X100 : Remplir le flacon
   RUNG wire#powerrail
      "X100_Remplir_DB"(OFF_SQ :=, INIT_SQ :=, ACK_EF :=, S_PREV :=, S_NEXT :=, SW_AUTO :=, SW_TAP :=, SW_TOP :=, SW_MAN :=, S_SEL :=, S_ON :=, S_OFF :=, T_PUSH :=, S_NO =>, S_MORE =>, S_ACTIVE =>, ERR_FLT =>, AUTO_ON =>, TAP_ON =>, TOP_ON =>, MAN_ON =>)
   END_RUNG
   // the same network as SCL:
   "X100_Remplir_DB"();   // "X100_Remplir"
END_REGION

REGION Network 4: X130 : Visser le bouchon sur le flacon
   RUNG wire#powerrail
      "X130_Visser_DB"(OFF_SQ :=, INIT_SQ :=, ACK_EF :=, S_PREV :=, S_NEXT :=, SW_AUTO :=, SW_TAP :=, SW_TOP :=, SW_MAN :=, S_SEL :=, S_ON :=, S_OFF :=, T_PUSH :=, S_NO =>, S_MORE =>, S_ACTIVE =>, ERR_FLT =>, AUTO_ON =>, TAP_ON =>, TOP_ON =>, MAN_ON =>)
   END_RUNG
   // the same network as SCL:
   "X130_Visser_DB"();   // "X130_Visser"
END_REGION

REGION Network 5: X160 : Evacuer les flacons en sortie
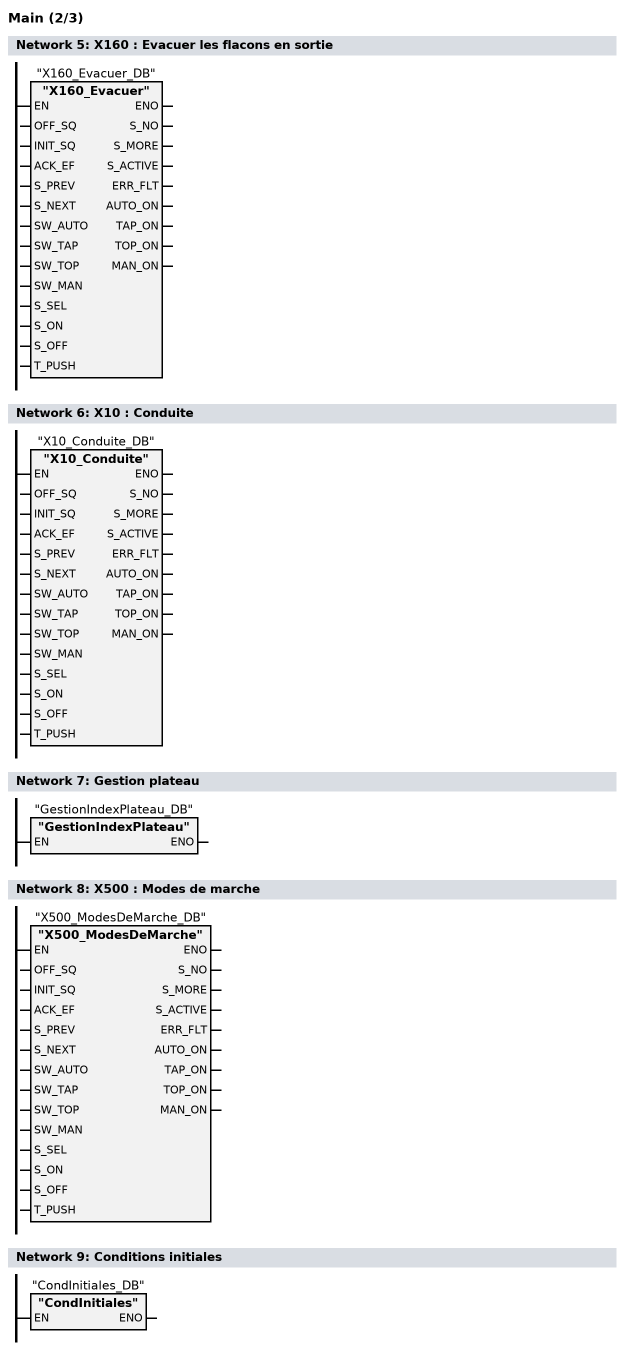
   RUNG wire#powerrail
      "X160_Evacuer_DB"(OFF_SQ :=, INIT_SQ :=, ACK_EF :=, S_PREV :=, S_NEXT :=, SW_AUTO :=, SW_TAP :=, SW_TOP :=, SW_MAN :=, S_SEL :=, S_ON :=, S_OFF :=, T_PUSH :=, S_NO =>, S_MORE =>, S_ACTIVE =>, ERR_FLT =>, AUTO_ON =>, TAP_ON =>, TOP_ON =>, MAN_ON =>)
   END_RUNG
   // the same network as SCL:
   "X160_Evacuer_DB"();   // "X160_Evacuer"
END_REGION

REGION Network 6: X10 : Conduite
   RUNG wire#powerrail
      "X10_Conduite_DB"(OFF_SQ :=, INIT_SQ :=, ACK_EF :=, S_PREV :=, S_NEXT :=, SW_AUTO :=, SW_TAP :=, SW_TOP :=, SW_MAN :=, S_SEL :=, S_ON :=, S_OFF :=, T_PUSH :=, S_NO =>, S_MORE =>, S_ACTIVE =>, ERR_FLT =>, AUTO_ON =>, TAP_ON =>, TOP_ON =>, MAN_ON =>)
   END_RUNG
   // the same network as SCL:
   "X10_Conduite_DB"();   // "X10_Conduite"
END_REGION

REGION Network 7: Gestion plateau
   RUNG wire#powerrail
      "GestionIndexPlateau_DB"()
   END_RUNG
   // the same network as SCL:
   "GestionIndexPlateau_DB"();   // "GestionIndexPlateau"
END_REGION

REGION Network 8: X500 : Modes de marche
   RUNG wire#powerrail
      "X500_ModesDeMarche_DB"(OFF_SQ :=, INIT_SQ :=, ACK_EF :=, S_PREV :=, S_NEXT :=, SW_AUTO :=, SW_TAP :=, SW_TOP :=, SW_MAN :=, S_SEL :=, S_ON :=, S_OFF :=, T_PUSH :=, S_NO =>, S_MORE =>, S_ACTIVE =>, ERR_FLT =>, AUTO_ON =>, TAP_ON =>, TOP_ON =>, MAN_ON =>)
   END_RUNG
   // the same network as SCL:
   "X500_ModesDeMarche_DB"();   // "X500_ModesDeMarche"
END_REGION

REGION Network 9: Conditions initiales
   RUNG wire#powerrail
      "CondInitiales_DB"()
   END_RUNG
   // the same network as SCL:
   "CondInitiales_DB"();   // "CondInitiales"
END_REGION

REGION Network 10
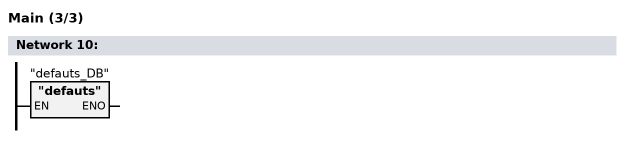
   RUNG wire#powerrail
      "defauts_DB"()
   END_RUNG
   // the same network as SCL:
   "defauts_DB"();   // "defauts"
END_REGION
END_ORGANIZATION_BLOCK